ABB RobotStudio station: ProyectoFinal2021-1.rspag

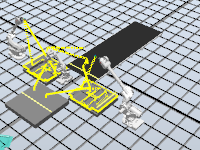
--- station ---
Station Station (saved by RobotStudio 20.4.9280.0)
Controller Controlador_Robot2, task T_ROB1: task frame (RAPID world) sits at (-153.05, 0, 0) mm in the station
Controller Controlador_Robot1, task T_ROB1: task frame (RAPID world) sits at (-2455.32, 2589.54, 0) mm in the station
Controller Controlador_PickPlace, task T_ROB1: task frame (RAPID world) sits at (-2646.21, -2443.71, 0) mm, rotated rx 0 ry 0 rz 90 deg in the station
Controller Controlador_PickPlace
  mechanical unit ROB_1: IRB6620_150_220__01, 6 joints, base frame (0, -2646.21, 459.11) mm
Controller Controlador_Robot1
  mechanical unit ROB_1: IRB7600_150_350__03, 6 joints, base frame (-2143.25, -4972.95, 0) mm
Controller Controlador_Robot2
  mechanical unit ROB_1: IRB7600_150_350__03_2, 6 joints, base frame (5003.05, -2378.13, 0) mm, rotated rx 0 ry 0 rz 180 deg
Layout (positions relative to the parent item):
  - Part Studio 3_2 [part] at (-2193.42, -2509.62, 250) mm, rotated rx 0 ry 0 rz 90 deg
  - IRB6620_150_220__01 [mechanism, from Robots\IRB6620_150_220_G_01.rslib] at (0, -2443.71, 459.11) mm, rotated rx 0 ry 0 rz 90 deg; joint values [1.5495, 0.9868, 0.0933, 0, 0.4907, -1.5921] (rad or m)
  - Vacuum Tool [mechanism] at (-1727.43, -2406.93, 788.65) mm, rotated rx 180 ry 0 rz 90 deg
      TCP tVacuum at (0, 0, 300) mm
      links: Vacuum Tool
  - Belt Conveyor [part] at (1369.01, -1300.28, 0) mm, rotated rx 0 ry 0 rz 90 deg
  - Componente inteligente_1 [smart component]
      signals: DI Attach, DI Dattach, DO Out_Sensor, DO Out_Sensor2, DO Out_Sensor22, DI AttR1, DI AttR2, DI DAttR1, DI DattR2, DO Out_Sensor5, DO Out_Sensor4, DO Out_Sensor6, DO Out_Sensor4_1, DO Out_Sensor_6_1
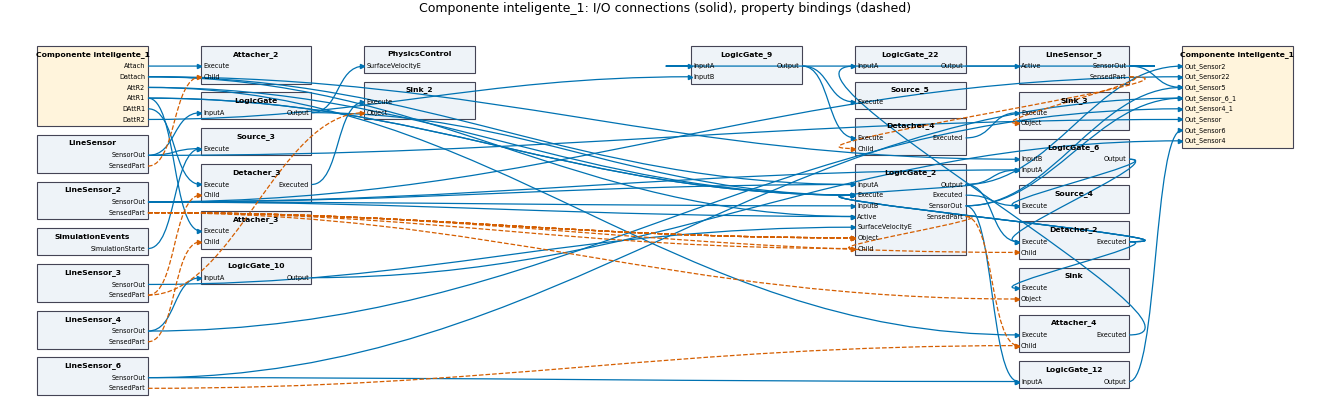
      connections:
        Componente inteligente_1.Attach -> Attacher_2.Execute
        LineSensor.SensorOut -> Source_3.Execute
        LogicGate.Output -> PhysicsControl.SurfaceVelocityEnabled
        Componente inteligente_1.Dattach -> LogicGate_2.InputA
        LogicGate_2.Output -> Detacher_2.Execute
        LogicGate.Output -> Positioner.Execute
        LineSensor_2.SensorOut -> LogicGate_3.InputB
        LogicGate_3.Output -> Positioner_2.Execute
        LogicGate_5.Output -> Componente inteligente_1.Out_Sensor2
        LineSensor_2.SensorOut -> LogicGate_5.InputA
        Detacher_2.Executed -> Positioner_3.Execute
        Detacher_2.Executed -> Positioner_4.Execute
        Componente inteligente_1.AttR2 -> Detacher_3.Execute
        Componente inteligente_1.AttR1 -> Attacher_3.Execute
        LineSensor_2.SensorOut -> Componente inteligente_1.Out_Sensor22
        Detacher_2.Executed -> Hide.Execute
        Componente inteligente_1.AttR1 -> Show.Execute
        Componente inteligente_1.Dattach -> LogicGate_6.InputB
        LogicGate_6.Output -> Detacher_2.Execute
        LineSensor_2.SensorOut -> Timer.Active
        Timer.Output -> LogicGate_6.InputA
        LineSensor_2.SensorOut -> LogicGate_6.InputA
        Hide_4.Executed -> Source_4.Execute
        Detacher_2.Executed -> Sink.Execute
        Componente inteligente_1.Dattach -> Timer_2.Active
        LogicGate_6.Output -> Source_4.Execute
        SimulationEvents.SimulationStarted -> Source_3.Execute
        Componente inteligente_1.AttR1 -> Attacher_3.Execute
        Componente inteligente_1.DAttR1 -> Detacher_3.Execute
        LineSensor_3.SensorOut -> PhysicsControl_2.SurfaceVelocityEnabled
        Detacher_3.Executed -> Sink_2.Execute
        LineSensor_5.SensorOut -> Componente inteligente_1.Out_Sensor5
        LineSensor_5.SensorOut -> Componente inteligente_1.Out_Sensor5
        LineSensor_5.SensorOut -> LogicGate_9.InputA
        Componente inteligente_1.DattR2 -> LogicGate_9.InputB
        LogicGate_9.Output -> Source_5.Execute
        LogicGate_9.Output -> Detacher_4.Execute
        Detacher_4.Executed -> Sink_3.Execute
        LineSensor_4.SensorOut -> LogicGate_10.InputA
        LineSensor_6.SensorOut -> LogicGate_12.InputA
        LineSensor_6.SensorOut -> Componente inteligente_1.Out_Sensor_6_1
        Componente inteligente_1.AttR2 -> Attacher_4.Execute
        LineSensor.SensorOut -> LogicGate.InputA
        LineSensor_6.SensorOut -> LogicGate_12.InputA
        LineSensor_6.SensorOut -> Componente inteligente_1.Out_Sensor_6_1
        LineSensor_4.SensorOut -> Componente inteligente_1.Out_Sensor4_1
        LineSensor.SensorOut -> Componente inteligente_1.Out_Sensor
        LogicGate_12.Output -> Componente inteligente_1.Out_Sensor6
        LogicGate_10.Output -> Componente inteligente_1.Out_Sensor4
        Attacher_4.Executed -> LogicGate_22.InputA
        LogicGate_22.Output -> LineSensor_5.Active
        LineSensor.SensedPart => Attacher_2.Child
        LineSensor_2.SensedPart => Detacher_2.Child
        LineSensor_2.SensedPart => Positioner.Object
        LineSensor_2.SensedPart => Positioner_2.Object
        LineSensor_2.SensedPart => Positioner_3.Object
        LineSensor_2.SensedPart => Positioner_4.Object
        LineSensor_2.SensedPart => Attacher_3.Child
        LineSensor_3.SensedPart => Detacher_3.Child
        LineSensor_2.SensedPart => Hide.Object
        LineSensor_2.SensedPart => Show.Object
        LineSensor_2.SensedPart => Sink.Object
        LineSensor_4.SensedPart => Attacher_3.Child
        LineSensor_3.SensedPart => Detacher_3.Child
        LineSensor_3.SensedPart => Sink_2.Object
        LineSensor_5.SensedPart => Detacher_4.Child
        LineSensor_5.SensedPart => Sink_3.Object
        LineSensor_6.SensedPart => Attacher_4.Child
        LineSensor_6.SensedPart => Attacher_4.Child
    - Detacher_2 [smart component, from Components\Detacher.rslib]
        properties: Child=(none); KeepPosition=true
    - Attacher_2 [smart component, from Components\Attacher.rslib]
        properties: Parent=Vacuum Tool; Flange=0; Child=(none); Mount=false; Offset=[0 0 0]; Orientation=[0 0 0]
    - LineSensor [smart component, from Components\LineSensor.rslib]
        properties: Start=[-1.2 -1 0.32]; End=[1.4 -1 0.32]; Radius=0.015; SensedPart=(none); SensedPoint=[-0.930547607421875 -1.00000006103516 0.32]
      - _sensorPart_ [part]
    - Source_3 [smart component, from Components\Source.rslib]
        properties: Source=Part Studio; Copy=(none); Parent=(none); Position=[-0.078281 5.030563 0.480363]; Orientation=[3.14159265358979 0 0]; Transient=true; PhysicsBehavior=3
    - SimulationEvents [smart component, from Components\SimulationEvents.rslib]
    - PhysicsControl [smart component, from Components\PhysicsControl.rslib]
        properties: Object=Belt Conveyor; Behavior=1; SurfaceVelocity=1
    - LogicGate [smart component, from Components\LogicGate.rslib]
        properties: Operator=NOT; Delay=0
    - LineSensor_2 [smart component, from Components\LineSensor.rslib]
        properties: Start=[-2.95 -1.5 0.533]; End=[-2.95 -3.2 0.533]; Radius=0.1; SensedPart=(none); SensedPoint=[-2.95000048828125 -1.55674926757812 0.533]
      - _sensorPart_ [part]
    - LogicGate_6 [smart component, from Components\LogicGate.rslib]
        properties: Operator=AND; Delay=1
    - Sink [smart component, from Components\Sink.rslib]
        properties: Object=(none)
    - Attacher_3 [smart component, from Components\Attacher.rslib]
        properties: Parent=Vacuum Tool; Flange=0; Child=(none); Mount=false; Offset=[0 0 0]; Orientation=[0 0 0]
    - Attacher_4 [smart component, from Components\Attacher.rslib]
        properties: Parent=Vacuum Tool; Flange=0; Child=(none); Mount=false; Offset=[0 0 0]; Orientation=[0 0 0]
    - Detacher_3 [smart component, from Components\Detacher.rslib]
        properties: Child=(none); KeepPosition=true
    - LineSensor_3 [smart component, from Components\LineSensor.rslib]
        properties: Start=[-1.2 -5 0.45]; End=[1.4 -5 0.45]; Radius=0.015; SensedPart=(none); SensedPoint=[0 0 0]
      - _sensorPart_ [part]
    - LineSensor_4 [smart component, from Components\LineSensor.rslib] at (1207.2, 0, 0) mm
        properties: Start=[-2.96159134746791 -3 0.312]; End=[-2.96159134746791 -2.881925 0.312]; Radius=0.001; SensedPart=(none); SensedPoint=[0 0 0]
      - _sensorPart_ [part]
    - Source_4 [smart component, from Components\Source.rslib]
        properties: Source=Part Studio_2; Copy=(none); Parent=(none); Position=[-1.791727 -2.471099 0.33]; Orientation=[3.14159265358979 0 1.5707963267949]; Transient=true; PhysicsBehavior=1
    - Sink_2 [smart component, from Components\Sink.rslib]
        properties: Object=(none)
    - Source_5 [smart component, from Components\Source.rslib]
        properties: Source=Part Studio_2; Copy=(none); Parent=(none); Position=[2.038141 -2.374172 0.33]; Orientation=[3.14159265358979 0 -1.5707963267949]; Transient=true; PhysicsBehavior=1
    - LineSensor_5 [smart component, from Components\LineSensor.rslib] at (6071.62, 0, 0) mm
        properties: Start=[-2.95 -1.5 0.533]; End=[-2.95 -3.2 0.533]; Radius=0.1; SensedPart=(none); SensedPoint=[0 0 0]
      - _sensorPart_ [part]
    - LogicGate_9 [smart component, from Components\LogicGate.rslib]
        properties: Operator=AND; Delay=0
    - Detacher_4 [smart component, from Components\Detacher.rslib]
        properties: Child=(none); KeepPosition=true
    - Sink_3 [smart component, from Components\Sink.rslib]
        properties: Object=(none)
    - LogicGate_10 [smart component, from Components\LogicGate.rslib]
        properties: Operator=NOT; Delay=0
    - LogicGate_12 [smart component, from Components\LogicGate.rslib]
        properties: Operator=NOT; Delay=0
    - LineSensor_6 [smart component, from Components\LineSensor.rslib] at (4964.36, 0, 0) mm
        properties: Start=[-2.96159134746791 -3 0.312]; End=[-2.96159134746791 -2.881925 0.312]; Radius=0.001; SensedPart=(none); SensedPoint=[2.0027666015625 -3 0.312]
      - _sensorPart_ [part]
    - LogicGate_22 [smart component, from Components\LogicGate.rslib]
        properties: Operator=NOT; Delay=0
  - Part Studio [part] at (384.19, -4809.35, 381.64) mm, rotated rx 180 ry 0 rz 0 deg
  - IRB7600_150_350__03 [mechanism, from Robots\IRB7600_150_350_G_03.rslib] at (-4598.56, -2383.41, 0) mm; joint values [0, -0.9152, 0, 0, 0.5236, 0] (rad or m)
  - LogicGate_7 [smart component, from Components\LogicGate.rslib]
      properties: Operator=AND; Delay=0
  - Pieza_1 [part] at (-1268.57, -2175.31, 0) mm
  - HerramientaDeCorte [mechanism, from Libraries\HerramientaDeCorte.rslib] at (-3713.92, -2383.41, 3226.26) mm, rotated rx 0 ry 67.56 rz 0 deg
  - Part Studio_2 [part] at (2038.14, -2374.17, 330) mm, rotated rx 180 ry 0 rz -90 deg
  - Part Studio 3_3 [part] at (2439.83, -2335.65, 250) mm, rotated rx 0 ry 0 rz -90 deg
  - IRB7600_150_350__03_2 [mechanism, from Robots\IRB7600_150_350_G_03.rslib] at (4850, -2378.13, 0) mm, rotated rx 0 ry 0 rz 180 deg; joint values [0, 0, -0.648, 0, 0.5236, 0] (rad or m)
  - HerramientaDeCorte_2 [mechanism, from Libraries\HerramientaDeCorte_1.rslib] at (2687.31, -2378.13, 3231.92) mm, rotated rx 0 ry 82.87 rz 180 deg
  - LogicGate_8 [smart component, from Components\LogicGate.rslib]
      properties: Operator=AND; Delay=0
  - LogicGate_11 [smart component, from Components\LogicGate.rslib]
      properties: Operator=AND; Delay=0
  - LogicGate_13 [smart component, from Components\LogicGate.rslib]
      properties: Operator=AND; Delay=0
  - LogicGate_14 [smart component, from Components\LogicGate.rslib]
      properties: Operator=AND; Delay=0
  - LogicGate_15 [smart component, from Components\LogicGate.rslib]
      properties: Operator=AND; Delay=0
  - LogicGate_16 [smart component, from Components\LogicGate.rslib]
      properties: Operator=AND; Delay=0
  - LogicGate_17 [smart component, from Components\LogicGate.rslib]
      properties: Operator=AND; Delay=0
  - LogicGate_18 [smart component, from Components\LogicGate.rslib]
      properties: Operator=AND; Delay=0
  - LogicGate_19 [smart component, from Components\LogicGate.rslib]
      properties: Operator=NOT; Delay=0
  - LogicGate_20 [smart component, from Components\LogicGate.rslib]
      properties: Operator=AND; Delay=0
  - LogicGate_21 [smart component, from Components\LogicGate.rslib]
      properties: Operator=NOT; Delay=0
  - Part Studio_291 [part] at (700.63, -8575.01, 80.62) mm, rotated rx -178.41 ry 0 rz 123.64 deg
Attachment: Vacuum Tool is attached to IRB6620_150_220__01 / Link6
Attachment: HerramientaDeCorte is attached to IRB7600_150_350__03 / Link6
Attachment: HerramientaDeCorte_2 is attached to IRB7600_150_350__03_2 / Link6
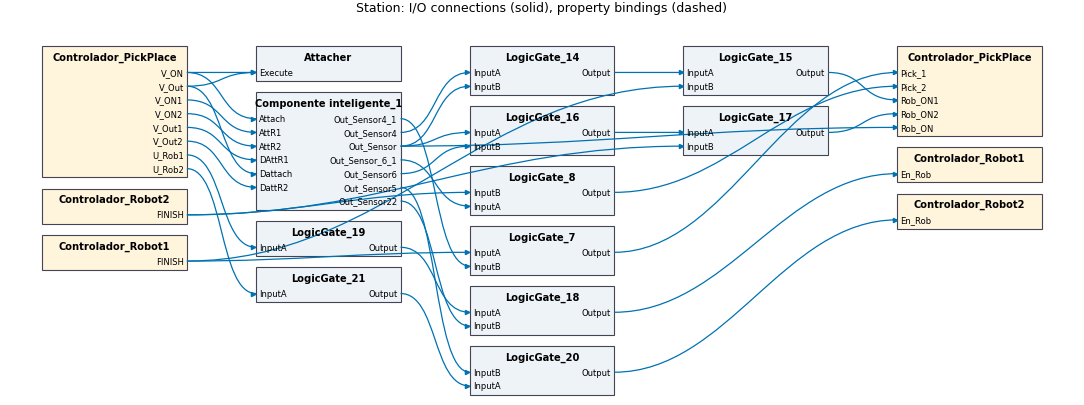
Station logic (signal -> signal, property => property):
  Controlador_PickPlace.V_ON -> Attacher.Execute
  Controlador_PickPlace.V_Out -> Detacher.Execute
  Controlador_PickPlace.V_ON -> Componente inteligente_1.Attach
  Controlador_PickPlace.V_ON1 -> Componente inteligente_1.AttR1
  Controlador_PickPlace.V_ON2 -> Componente inteligente_1.AttR2
  Controlador_PickPlace.V_Out1 -> Componente inteligente_1.DAttR1
  Controlador_PickPlace.V_Out -> Componente inteligente_1.Dattach
  Controlador_Robot2.FINISH -> LogicGate_8.InputB
  Controlador_PickPlace.V_Out2 -> Componente inteligente_1.DattR2
  Controlador_Robot1.FINISH -> LogicGate_7.InputA
  Componente inteligente_1.Out_Sensor4_1 -> LogicGate_7.InputB
  Componente inteligente_1.Out_Sensor4 -> LogicGate_14.InputA
  Componente inteligente_1.Out_Sensor -> LogicGate_14.InputB
  LogicGate_14.Output -> LogicGate_15.InputA
  Controlador_Robot1.FINISH -> LogicGate_15.InputB
  LogicGate_7.Output -> Controlador_PickPlace.Pick_1
  Componente inteligente_1.Out_Sensor_6_1 -> LogicGate_8.InputA
  LogicGate_8.Output -> Controlador_PickPlace.Pick_2
  Componente inteligente_1.Out_Sensor -> LogicGate_16.InputA
  Componente inteligente_1.Out_Sensor6 -> LogicGate_16.InputB
  LogicGate_16.Output -> LogicGate_17.InputA
  Controlador_Robot2.FINISH -> LogicGate_17.InputB
  LogicGate_15.Output -> Controlador_PickPlace.Rob_ON1
  LogicGate_17.Output -> Controlador_PickPlace.Rob_ON2
  Componente inteligente_1.Out_Sensor -> Controlador_PickPlace.Rob_ON
  Controlador_PickPlace.U_Rob1 -> LogicGate_19.InputA
  LogicGate_19.Output -> LogicGate_18.InputA
  LogicGate_18.Output -> Controlador_Robot1.En_Rob
  Controlador_PickPlace.U_Rob2 -> LogicGate_21.InputA
  Componente inteligente_1.Out_Sensor5 -> LogicGate_20.InputB
  LogicGate_21.Output -> LogicGate_20.InputA
  LogicGate_20.Output -> Controlador_Robot2.En_Rob
  Componente inteligente_1.Out_Sensor22 -> LogicGate_18.InputB
Targets, tools, work objects and paths stored in the station and not in the controller backup, written as RAPID:
! task T_ROB1
MODULE Module1
  CONST robtarget Target_274:=[[250.928875654,-5796.464620021,317.65],[0,-0.707106781,0.707106781,0],[-1,0,-2,0],[9E+09,9E+09,9E+09,9E+09,9E+09,9E+09]];
  CONST robtarget Target_404:=[[700.928875654,-5166.464620021,352.65],[0,-0.707106781,0.707106781,0],[-1,0,-2,0],[9E+09,9E+09,9E+09,9E+09,9E+09,9E+09]];
  CONST robtarget Target_444:=[[700.928875654,-4846.464620021,352.65],[0,-0.707106781,0.707106781,0],[0,0,-1,0],[9E+09,9E+09,9E+09,9E+09,9E+09,9E+09]];
ENDMODULE


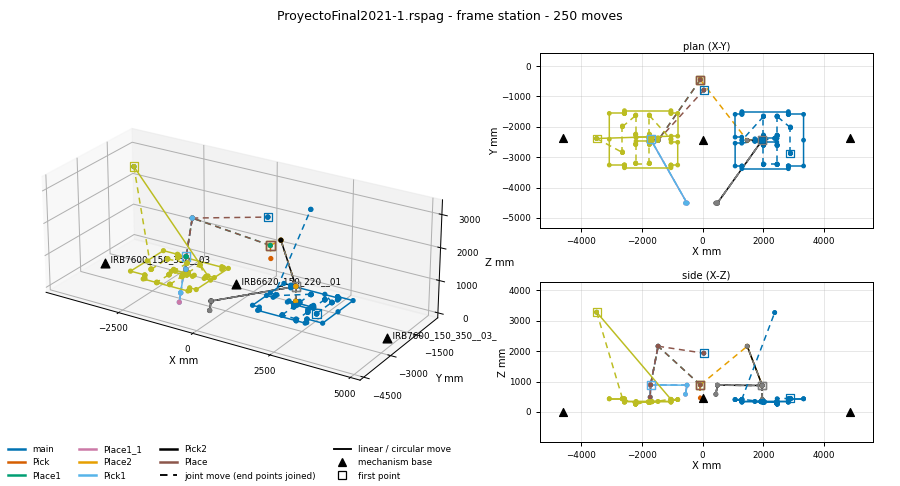
[picture p0: tool path of ProyectoFinal2021-1.rspag in frame station, 250 of 250 moves have a stored position in this frame; points joined in program order, loops and branches not executed]
--- Backups/Controlador_PickPlace/RAPID/TASK1/PROGMOD/CalibData.mod ---
MODULE CalibData
    PERS tooldata tVacuum:=[TRUE,[[0,0,300],[1,0,0,0]],[11,[0,0,200],[1,0,0,0],0,0,0]];
ENDMODULE

--- Backups/Controlador_PickPlace/RAPID/TASK1/PROGMOD/Module1.mod ---
MODULE Module1
        CONST robtarget Target_10:=[[0,-1179.406420384,2164.113508615],[0.353553391,-0.612372436,0.612372436,0.353553391],[0,-1,0,0],[9E+09,9E+09,9E+09,9E+09,9E+09,9E+09]];
    CONST robtarget Target_20_2:=[[1993.099436165,-2567.929041541,890],[0,-0.707106781,0.707106781,0],[-1,0,-1,0],[9E+09,9E+09,9E+09,9E+09,9E+09,9E+09]];
    CONST robtarget Target_20:=[[2025.267436165,-2567.931041541,460.348],[0,-0.707106781,0.707106781,0],[-2,0,-2,0],[9E+09,9E+09,9E+09,9E+09,9E+09,9E+09]];
    CONST robtarget Target_30_2:=[[36.785436165,-931.826041541,890],[0,1,0,0],[-1,0,-2,0],[9E+09,9E+09,9E+09,9E+09,9E+09,9E+09]];
    CONST robtarget Target_30:=[[36.785436165,-918.776041541,488.65],[0,1,0,0],[-1,0,-2,0],[9E+09,9E+09,9E+09,9E+09,9E+09,9E+09]];
    CONST robtarget Target_30_3:=[[2015.725,-2164.754477706,320.279],[0,-0.707106781,0.707106781,0],[0,0,-1,0],[9E+09,9E+09,9E+09,9E+09,9E+09,9E+09]];
    CONST robtarget Target_40:=[[-2065.640563835,-2080.403041541,581.641],[0,-0.707106781,0.707106781,0],[0,0,0,0],[9E+09,9E+09,9E+09,9E+09,9E+09,9E+09]];
    CONST robtarget Target_50:=[[5.364436165,-4607.016041541,411.65],[0,0,1,0],[-1,0,-1,0],[9E+09,9E+09,9E+09,9E+09,9E+09,9E+09]];
    CONST robtarget Target_60:=[[0,-4113.021984806,2164.113532469],[0.353553384,0.612372439,0.612372439,-0.353553384],[-2,0,-1,0],[9E+09,9E+09,9E+09,9E+09,9E+09,9E+09]];
    CONST robtarget Target_70:=[[1653.263,-2683.789477706,1934.535],[0,-0.707106781,0.707106781,0],[-1,0,-2,0],[9E+09,9E+09,9E+09,9E+09,9E+09,9E+09]];
    CONST robtarget Target_80:=[[-2065.640563835,-3080.403041541,581.641],[0,1,0,0],[-2,0,-1,0],[9E+09,9E+09,9E+09,9E+09,9E+09,9E+09]];
    CONST robtarget Target_90:=[[1653.26,-2638.786477706,434.509],[0,-0.707106781,0.707106781,0],[0,0,-1,0],[9E+09,9E+09,9E+09,9E+09,9E+09,9E+09]];
    CONST robtarget Target_100:=[[1553.362,-2638.786477706,441.414],[0,-0.707106781,0.707106781,0],[0,0,-1,0],[9E+09,9E+09,9E+09,9E+09,9E+09,9E+09]];
    CONST robtarget Target_110:=[[1453.462,-2638.788477706,448.319],[0,-0.707106781,0.707106781,0],[0,0,-1,0],[9E+09,9E+09,9E+09,9E+09,9E+09,9E+09]];
    CONST robtarget Target_120:=[[1453.471,-2728.784477706,448.368],[0,-0.707106781,0.707106781,0],[-1,0,-2,0],[9E+09,9E+09,9E+09,9E+09,9E+09,9E+09]];
    CONST robtarget Target_40_2:=[[-2065.640563835,-2130.403041541,881.641],[0,-0.707106781,0.707106781,0],[0,0,0,0],[9E+09,9E+09,9E+09,9E+09,9E+09,9E+09]];
    CONST robtarget Target_50_2:=[[5.364436165,-4607.016041541,871.65],[0,0,1,0],[-1,0,-1,0],[9E+09,9E+09,9E+09,9E+09,9E+09,9E+09]];
    CONST robtarget Target_80_2:=[[-2065.640563835,-3130.403041541,881.641],[0,1,0,0],[-2,0,-1,0],[9E+09,9E+09,9E+09,9E+09,9E+09,9E+09]];
!***********************************************************
    !
    ! Módulo:  Module1
    !
    ! Descripción:
    !   <Introduzca la descripción aquí>
    !
    ! Autor: Alex
    !
    ! Versión: 1.0
    !
    !***********************************************************


    !***********************************************************
    !
    ! Procedimiento Main
    !
    !   Este es el punto de entrada de su programa
    !
    !***********************************************************
    PROC main()
        Init:
        SetDO V_Out,0;
        SetDO V_ON,0;
        SetDO U_Rob1,0;
        SetDO U_Rob2,0;
        MoveJ Target_70,v1000,z100,tVacuum\WObj:=wobj0;
        WaitDI Rob_ON,1;
 !       WaitUntil Rob_ON1=1 OR Rob_ON2=1 OR Pick_1=1 OR Pick_2=1 OR Rob_ON1=0 OR Rob_ON2=0 OR Pick_1=0 OR Pick_2=0;
        IF Rob_ON1=1 THEN ! Detecta si robot está quieto, hay tapete esperando y no hay tapete en estación 1, pone tapete en estación 1
           pick;
           place1;
        ELSEIF Rob_ON2=1 THEN ! Detecta si robot está quieto, hay tapete esperando y no hay tapete en estación 2, pone tapete en estación 2
           pick;
           place2;
        ELSEIF Pick_1=1 THEN !Detecta si robot 1 está quieto y hay tapete en estación 1, lleva el tapete de estación 1 a mesa
           pick1;
        ELSEIF Pick_2=1 THEN !Detecta si robot 2 está quieto y hay tapete en estación 2, lleva el tapete de estación 2 a mesa
           pick2;
        ELSE MoveJ Target_70,v1000,fine,tVacuum\WObj:=wobj0;
        ENDIF
        GOTO Init;
        !Añada aquí su código
    ENDPROC
    PROC Pick()
        MoveJ Target_20_2,v1000,fine,tVacuum\WObj:=wobj0;
        MoveJ Target_20,v1000,fine,tVacuum\WObj:=wobj0;
        WaitTime 1;
        SetDO V_ON,1;
        WaitTime 2;
        SetDO V_ON,0;
    ENDPROC
    PROC Place1()
        MoveJ Target_20_2,v1000,fine,tVacuum\WObj:=wobj0;
        MoveJ Target_10,v1000,fine,tVacuum\WObj:=wobj0;
        MoveJ Target_30_2,v1000,fine,tVacuum\WObj:=wobj0;
        MoveJ Target_30,v1000,fine,tVacuum\WObj:=wobj0;
        WaitTime 1;
        SetDO V_Out,1;
        WaitTime 1;
        SetDO V_Out,0;
        MoveJ Target_30_2,v1000,fine,tVacuum\WObj:=wobj0;
        MoveJ Target_10,v1000,fine,tVacuum\WObj:=wobj0;
    ENDPROC
    PROC Place1_1()
        MoveJ Target_30_2,v1000,fine,tVacuum\WObj:=wobj0;
        WaitTime 1;
        MoveJ Target_30,v1000,fine,tVacuum\WObj:=wobj0;
        SetDO V_ON1,1;
        WaitTime 1;
        SetDO V_ON1,0;
        MoveJ Target_30_2,v1000,fine,tVacuum\WObj:=wobj0;
        MoveJ Target_40_2,v1000,fine,tVacuum\WObj:=wobj0;
        MoveJ Target_40,v1000,fine,tVacuum\WObj:=wobj0;
        SetDO V_Out1,1;
        WaitTime 1;
        SetDO V_Out1,0;
        MoveJ Target_40_2,v1000,fine,tVacuum\WObj:=wobj0;
        MoveJ Target_30_2,v1000,fine,tVacuum\WObj:=wobj0;
        MoveJ Target_10,v1000,fine,tVacuum\WObj:=wobj0;
    ENDPROC
    PROC Place2()
        MoveJ Target_20_2,v1000,fine,tVacuum\WObj:=wobj0;
        MoveJ Target_60,v1000,fine,tVacuum\WObj:=wobj0;
        MoveJ Target_50_2,v1000,fine,tVacuum\WObj:=wobj0;
        WaitTime 1;
        MoveJ Target_50,v1000,fine,tVacuum\WObj:=wobj0;
        WaitTime 1;
        SetDO V_Out2,1;
        WaitTime 1;
        SetDO V_Out2,0;
        MoveJ Target_50_2,v1000,fine,tVacuum\WObj:=wobj0;
        MoveJ Target_60,v1000,fine,tVacuum\WObj:=wobj0;
    ENDPROC
    PROC Pick1()
        MoveL Target_30_2,v1000,fine,tVacuum\WObj:=wobj0;
        MoveL Target_30,v1000,fine,tVacuum\WObj:=wobj0;
        SetDO V_ON1,1;
        WaitTime 2;
        SetDO V_ON1,0;
        SetDO U_Rob1,1;
        MoveL Target_30_2,v1000,fine,tVacuum\WObj:=wobj0;
        MoveL Target_40_2,v1000,fine,tVacuum\WObj:=wobj0;
        MoveL Target_40,v1000,fine,tVacuum\WObj:=wobj0;
        SetDO V_Out1,1;
        WaitTime 2;
        SetDO V_Out1,0;
        WaitTime 2;
        SetDO U_Rob1,0;
        MoveJ Target_40_2,v1000,fine,tVacuum\WObj:=wobj0;
        MoveJ Target_30_2,v1000,fine,tVacuum\WObj:=wobj0;
        MoveJ Target_10,v1000,fine,tVacuum\WObj:=wobj0;
    ENDPROC
    PROC Pick2()
        MoveJ Target_50_2,v1000,fine,tVacuum\WObj:=wobj0;
        MoveJ Target_50,v1000,fine,tVacuum\WObj:=wobj0;
        SetDO V_ON2,1;
        WaitTime 2;
        SetDO V_ON2,0;
        WaitTime 2;
        SetDO U_Rob2,1;
        MoveJ Target_50_2,v1000,fine,tVacuum\WObj:=wobj0;
        MoveJ Target_80_2,v1000,fine,tVacuum\WObj:=wobj0;
        MoveJ Target_80,v1000,fine,tVacuum\WObj:=wobj0;
        SetDO V_Out1,1;
        WaitTime 2;
        SetDO V_Out1,0;
        WaitTime 2;
        SetDO U_Rob2,0;
        MoveL Target_80_2,v1000,fine,tVacuum\WObj:=wobj0;
        MoveL Target_50_2,v1000,fine,tVacuum\WObj:=wobj0;
        MoveL Target_60,v1000,fine,tVacuum\WObj:=wobj0;
    ENDPROC
    PROC Place()
        MoveJ Target_20_2,v1000,fine,tVacuum\WObj:=wobj0;
        MoveJ Target_10,v1000,fine,tVacuum\WObj:=wobj0;
        MoveJ Target_30_2,v1000,fine,tVacuum\WObj:=wobj0;
        MoveJ Target_30,v1000,fine,tVacuum\WObj:=wobj0;
        WaitTime 1;
        SetDO V_Out,1;
        WaitTime 1;
        SetDO V_Out,0;
        MoveJ Target_30_2,v1000,fine,tVacuum\WObj:=wobj0;
        MoveJ Target_10,v1000,fine,tVacuum\WObj:=wobj0;
        MoveJ Target_70,v1000,fine,tVacuum\WObj:=wobj0;
    ENDPROC
    PROC Place2_1()
        MoveJ Target_50_2,v1000,fine,tVacuum\WObj:=wobj0;
        MoveJ Target_50,v1000,fine,tVacuum\WObj:=wobj0;
        SetDO V_ON2,1;
        WaitTime 2;
        SetDO V_ON2,0;
        MoveJ Target_50_2,v1000,fine,tVacuum\WObj:=wobj0;
        MoveJ Target_80_2,v1000,fine,tVacuum\WObj:=wobj0;
        MoveJ Target_80,v1000,fine,tVacuum\WObj:=wobj0;
        SetDO V_out1,1;
        WaitTime 2;
        SetDO V_Out1,0;
        MoveJ Target_80_2,v1000,fine,tVacuum\WObj:=wobj0;
        MoveJ Target_50_2,v1000,fine,tVacuum\WObj:=wobj0;
        MoveJ Target_60,v1000,fine,tVacuum\WObj:=wobj0;
    ENDPROC

ENDMODULE

--- Backups/Controlador_Robot1/RAPID/TASK1/PROGMOD/CalibData.mod ---
MODULE CalibData
    PERS tooldata MyTool:=[TRUE,[[31.7926,0,229.639],[0.945519,0,0.325568,0]],[1,[0,0,1],[1,0,0,0],0,0,0]];
    PERS tooldata HerramientaDeCorte:=[TRUE,[[0,0,319.427],[1,0,0,0]],[1,[0,0,1],[1,0,0,0],0,0,0]];
ENDMODULE

--- Backups/Controlador_Robot1/RAPID/TASK1/PROGMOD/Module1.mod ---
MODULE Module1
        CONST robtarget Target_10:=[[783.928875653,-4994.669620021,486.089],[0,-0.707106781,0.707106781,0],[0,0,0,0],[9E+09,9E+09,9E+09,9E+09,9E+09,9E+09]];
    CONST robtarget Target_20:=[[740.928875653,-4996.464620021,391.65],[0,-0.707106781,0.707106781,0],[0,0,-1,0],[9E+09,9E+09,9E+09,9E+09,9E+09,9E+09]];
    CONST robtarget Target_10_2:=[[783.928875653,-4994.669620021,936.089],[0,-0.707106781,0.707106781,0],[0,0,-1,0],[9E+09,9E+09,9E+09,9E+09,9E+09,9E+09]];
    CONST robtarget Target_30:=[[-1034.222247941,-4972.95221081,3284.527172221],[0.604871201,0,0.79632332,0],[-1,0,-1,0],[9E+09,9E+09,9E+09,9E+09,9E+09,9E+09]];
    CONST robtarget Target_20_3:=[[740.928875653,-4996.464620021,451.65],[0,-0.707106781,0.707106781,0],[0,0,-1,0],[9E+09,9E+09,9E+09,9E+09,9E+09,9E+09]];
        TASK PERS tooldata tool1:=[TRUE,[[0,0,0],[1,0,0,0]],[-1,[0,0,0],[1,0,0,0],0,0,0]];
    CONST robtarget Target_35:=[[-186.231124346,-5433.964620021,446.65],[0,-0.707106781,0.707106781,0],[-1,0,-2,0],[9E+09,9E+09,9E+09,9E+09,9E+09,9E+09]];
    CONST robtarget Target_40:=[[-186.231124346,-5433.964620021,432.65],[0,-0.707106781,0.707106781,0],[-1,0,-2,0],[9E+09,9E+09,9E+09,9E+09,9E+09,9E+09]];
    CONST robtarget Target_50:=[[-173.731124346,-5421.464620021,432.65],[0,-0.707106781,0.707106781,0],[-1,0,-2,0],[9E+09,9E+09,9E+09,9E+09,9E+09,9E+09]];
    CONST robtarget Target_60:=[[-186.231124346,-5408.964620021,432.65],[0,-0.707106781,0.707106781,0],[-1,0,-2,0],[9E+09,9E+09,9E+09,9E+09,9E+09,9E+09]];
    CONST robtarget Target_70:=[[-198.731124346,-5421.464620021,432.65],[0,-0.707106781,0.707106781,0],[-1,0,-2,0],[9E+09,9E+09,9E+09,9E+09,9E+09,9E+09]];
    CONST robtarget Target_90:=[[-173.731124346,-4571.464620021,432.65],[0,-0.707106781,0.707106781,0],[0,0,0,0],[9E+09,9E+09,9E+09,9E+09,9E+09,9E+09]];
    CONST robtarget Target_110:=[[-198.731124346,-4571.464620021,432.65],[0,-0.707106781,0.707106781,0],[0,0,0,0],[9E+09,9E+09,9E+09,9E+09,9E+09,9E+09]];
    CONST robtarget Target_114:=[[250.928875654,-4216.464620021,437.65],[0,-0.707106781,0.707106781,0],[0,0,-1,0],[9E+09,9E+09,9E+09,9E+09,9E+09,9E+09]];
    CONST robtarget Target_115:=[[250.928875654,-4216.464620021,277.65],[0,-0.707106781,0.707106781,0],[0,0,0,0],[9E+09,9E+09,9E+09,9E+09,9E+09,9E+09]];
    CONST robtarget Target_120:=[[250.928875654,-4216.464620021,262.65],[0,-0.707106781,0.707106781,0],[0,0,0,0],[9E+09,9E+09,9E+09,9E+09,9E+09,9E+09]];
    CONST robtarget Target_130:=[[260.928875654,-4206.464620021,262.65],[0,-0.707106781,0.707106781,0],[0,0,0,0],[9E+09,9E+09,9E+09,9E+09,9E+09,9E+09]];
    CONST robtarget Target_140:=[[250.928875654,-4196.464620021,262.65],[0,-0.707106781,0.707106781,0],[0,0,0,0],[9E+09,9E+09,9E+09,9E+09,9E+09,9E+09]];
    CONST robtarget Target_150:=[[240.928875654,-4206.464620021,262.65],[0,-0.707106781,0.707106781,0],[0,0,0,0],[9E+09,9E+09,9E+09,9E+09,9E+09,9E+09]];
    CONST robtarget Target_155:=[[250.928875654,-4846.464620021,277.65],[0,-0.707106781,0.707106781,0],[0,0,0,0],[9E+09,9E+09,9E+09,9E+09,9E+09,9E+09]];
    CONST robtarget Target_160:=[[250.928875654,-4846.464620021,262.65],[0,-0.707106781,0.707106781,0],[0,0,0,0],[9E+09,9E+09,9E+09,9E+09,9E+09,9E+09]];
    CONST robtarget Target_170:=[[260.928875654,-4836.464620021,262.65],[0,-0.707106781,0.707106781,0],[0,0,0,0],[9E+09,9E+09,9E+09,9E+09,9E+09,9E+09]];
    CONST robtarget Target_180:=[[250.928875654,-4826.464620021,262.65],[0,-0.707106781,0.707106781,0],[0,0,0,0],[9E+09,9E+09,9E+09,9E+09,9E+09,9E+09]];
    CONST robtarget Target_190:=[[240.928875654,-4836.464620021,262.65],[0,-0.707106781,0.707106781,0],[0,0,0,0],[9E+09,9E+09,9E+09,9E+09,9E+09,9E+09]];
    CONST robtarget Target_195:=[[261.901875654,-4932.290620021,347.65],[0,-0.707106781,0.707106781,0],[0,0,0,0],[9E+09,9E+09,9E+09,9E+09,9E+09,9E+09]];
    CONST robtarget Target_200:=[[261.901875654,-4932.290620021,332.65],[0,-0.707106781,0.707106781,0],[0,0,0,0],[9E+09,9E+09,9E+09,9E+09,9E+09,9E+09]];
    CONST robtarget Target_210:=[[261.901875654,-5060.638620021,332.65],[0,-0.707106781,0.707106781,0],[-1,0,-2,0],[9E+09,9E+09,9E+09,9E+09,9E+09,9E+09]];
    CONST robtarget Target_220:=[[663.589875654,-5060.638620021,332.65],[0,-0.707106781,0.707106781,0],[-1,0,-2,0],[9E+09,9E+09,9E+09,9E+09,9E+09,9E+09]];
    CONST robtarget Target_230:=[[663.589875654,-4932.290620021,332.65],[0,-0.707106781,0.707106781,0],[0,0,0,0],[9E+09,9E+09,9E+09,9E+09,9E+09,9E+09]];
    CONST robtarget Target_234:=[[250.928875654,-5166.464620021,362.65],[0,-0.707106781,0.707106781,0],[-1,0,-2,0],[9E+09,9E+09,9E+09,9E+09,9E+09,9E+09]];
    CONST robtarget Target_235:=[[250.928875654,-5166.464620021,277.65],[0,-0.707106781,0.707106781,0],[-1,0,-2,0],[9E+09,9E+09,9E+09,9E+09,9E+09,9E+09]];
    CONST robtarget Target_240:=[[250.928875654,-5166.464620021,262.65],[0,-0.707106781,0.707106781,0],[-1,0,-2,0],[9E+09,9E+09,9E+09,9E+09,9E+09,9E+09]];
    CONST robtarget Target_250:=[[260.928875654,-5156.464620021,262.65],[0,-0.707106781,0.707106781,0],[-1,0,-2,0],[9E+09,9E+09,9E+09,9E+09,9E+09,9E+09]];
    CONST robtarget Target_260:=[[250.928875654,-5146.464620021,262.65],[0,-0.707106781,0.707106781,0],[-1,0,-2,0],[9E+09,9E+09,9E+09,9E+09,9E+09,9E+09]];
    CONST robtarget Target_270:=[[240.928875654,-5156.464620021,262.65],[0,-0.707106781,0.707106781,0],[-1,0,-2,0],[9E+09,9E+09,9E+09,9E+09,9E+09,9E+09]];
    CONST robtarget Target_275:=[[250.928875654,-5796.464620021,277.65],[0,-0.707106781,0.707106781,0],[-1,0,-2,0],[9E+09,9E+09,9E+09,9E+09,9E+09,9E+09]];
    CONST robtarget Target_280:=[[250.928875654,-5796.464620021,262.65],[0,-0.707106781,0.707106781,0],[-1,0,-2,0],[9E+09,9E+09,9E+09,9E+09,9E+09,9E+09]];
    CONST robtarget Target_290:=[[260.928875654,-5786.464620021,262.65],[0,-0.707106781,0.707106781,0],[-1,0,-2,0],[9E+09,9E+09,9E+09,9E+09,9E+09,9E+09]];
    CONST robtarget Target_300:=[[250.928875654,-5776.464620021,262.65],[0,-0.707106781,0.707106781,0],[-1,0,-2,0],[9E+09,9E+09,9E+09,9E+09,9E+09,9E+09]];
    CONST robtarget Target_310:=[[240.928875654,-5786.464620021,262.65],[0,-0.707106781,0.707106781,0],[-1,0,-2,0],[9E+09,9E+09,9E+09,9E+09,9E+09,9E+09]];
    CONST robtarget Target_325:=[[700.928875654,-5796.464620021,327.65],[0,-0.707106781,0.707106781,0],[-1,0,-2,0],[9E+09,9E+09,9E+09,9E+09,9E+09,9E+09]];
    CONST robtarget Target_330:=[[700.928875654,-5796.464620021,312.65],[0,-0.707106781,0.707106781,0],[-1,0,-2,0],[9E+09,9E+09,9E+09,9E+09,9E+09,9E+09]];
    CONST robtarget Target_340:=[[710.928875654,-5786.464620021,312.65],[0,-0.707106781,0.707106781,0],[-1,0,-2,0],[9E+09,9E+09,9E+09,9E+09,9E+09,9E+09]];
    CONST robtarget Target_350:=[[700.928875654,-5776.464620021,312.65],[0,-0.707106781,0.707106781,0],[-1,0,-2,0],[9E+09,9E+09,9E+09,9E+09,9E+09,9E+09]];
    CONST robtarget Target_360:=[[690.928875654,-5786.464620021,312.65],[0,-0.707106781,0.707106781,0],[-1,0,-2,0],[9E+09,9E+09,9E+09,9E+09,9E+09,9E+09]];
    CONST robtarget Target_365:=[[700.928875654,-5166.464620021,327.65],[0,-0.707106781,0.707106781,0],[-1,0,-2,0],[9E+09,9E+09,9E+09,9E+09,9E+09,9E+09]];
    CONST robtarget Target_370:=[[700.928875654,-5166.464620021,312.65],[0,-0.707106781,0.707106781,0],[-1,0,-2,0],[9E+09,9E+09,9E+09,9E+09,9E+09,9E+09]];
    CONST robtarget Target_380:=[[710.928875654,-5156.464620021,312.65],[0,-0.707106781,0.707106781,0],[-1,0,-2,0],[9E+09,9E+09,9E+09,9E+09,9E+09,9E+09]];
    CONST robtarget Target_390:=[[700.928875654,-5146.464620021,312.65],[0,-0.707106781,0.707106781,0],[-1,0,-2,0],[9E+09,9E+09,9E+09,9E+09,9E+09,9E+09]];
    CONST robtarget Target_400:=[[690.928875654,-5156.464620021,312.65],[0,-0.707106781,0.707106781,0],[-1,0,-2,0],[9E+09,9E+09,9E+09,9E+09,9E+09,9E+09]];
    CONST robtarget Target_405:=[[783.642875654,-5041.464620021,349.902],[0,-0.707106781,0.707106781,0],[-1,0,-2,0],[9E+09,9E+09,9E+09,9E+09,9E+09,9E+09]];
    CONST robtarget Target_410:=[[783.642875654,-5041.464620021,334.902],[0,-0.707106781,0.707106781,0],[-1,0,-2,0],[9E+09,9E+09,9E+09,9E+09,9E+09,9E+09]];
    CONST robtarget Target_420:=[[983.642875654,-5041.464620021,345.449],[0,-0.707106781,0.707106781,0],[-1,0,-2,0],[9E+09,9E+09,9E+09,9E+09,9E+09,9E+09]];
    CONST robtarget Target_430:=[[983.642875654,-4951.464620021,345.449],[0,-0.707106781,0.707106781,0],[0,0,0,0],[9E+09,9E+09,9E+09,9E+09,9E+09,9E+09]];
    CONST robtarget Target_440:=[[783.642875654,-4951.464620021,334.902],[0,-0.707106781,0.707106781,0],[0,0,0,0],[9E+09,9E+09,9E+09,9E+09,9E+09,9E+09]];
    CONST robtarget Target_445:=[[700.928875654,-4846.464620021,327.65],[0,-0.707106781,0.707106781,0],[0,0,0,0],[9E+09,9E+09,9E+09,9E+09,9E+09,9E+09]];
    CONST robtarget Target_450:=[[700.928875654,-4846.464620021,312.65],[0,-0.707106781,0.707106781,0],[0,0,0,0],[9E+09,9E+09,9E+09,9E+09,9E+09,9E+09]];
    CONST robtarget Target_460:=[[710.928875654,-4836.464620021,312.65],[0,-0.707106781,0.707106781,0],[0,0,0,0],[9E+09,9E+09,9E+09,9E+09,9E+09,9E+09]];
    CONST robtarget Target_470:=[[700.928875654,-4826.464620021,312.65],[0,-0.707106781,0.707106781,0],[0,0,0,0],[9E+09,9E+09,9E+09,9E+09,9E+09,9E+09]];
    CONST robtarget Target_480:=[[690.928875654,-4836.464620021,312.65],[0,-0.707106781,0.707106781,0],[0,0,0,0],[9E+09,9E+09,9E+09,9E+09,9E+09,9E+09]];
    CONST robtarget Target_485:=[[700.928875654,-4216.464620021,327.65],[0,-0.707106781,0.707106781,0],[0,0,0,0],[9E+09,9E+09,9E+09,9E+09,9E+09,9E+09]];
    CONST robtarget Target_490:=[[700.928875654,-4216.464620021,312.65],[0,-0.707106781,0.707106781,0],[0,0,0,0],[9E+09,9E+09,9E+09,9E+09,9E+09,9E+09]];
    CONST robtarget Target_500:=[[710.928875654,-4206.464620021,312.65],[0,-0.707106781,0.707106781,0],[0,0,0,0],[9E+09,9E+09,9E+09,9E+09,9E+09,9E+09]];
    CONST robtarget Target_510:=[[700.928875654,-4196.464620021,312.65],[0,-0.707106781,0.707106781,0],[0,0,0,0],[9E+09,9E+09,9E+09,9E+09,9E+09,9E+09]];
    CONST robtarget Target_520:=[[690.928875654,-4206.464620021,312.65],[0,-0.707106781,0.707106781,0],[0,0,0,0],[9E+09,9E+09,9E+09,9E+09,9E+09,9E+09]];
    CONST robtarget Target_530:=[[-963.36800286,-4972.95221081,3348.184668964],[0.831174335,0,0.556011892,0],[-1,0,-1,0],[9E+09,9E+09,9E+09,9E+09,9E+09,9E+09]];
    CONST robtarget Target_194:=[[240.928875654,-4836.464620021,347.65],[0,-0.707106781,0.707106781,0],[0,0,-1,0],[9E+09,9E+09,9E+09,9E+09,9E+09,9E+09]];
    CONST robtarget Target_75:=[[-186.231124346,-4583.964620021,446.65],[0,-0.707106781,0.707106781,0],[0,0,-1,0],[9E+09,9E+09,9E+09,9E+09,9E+09,9E+09]];
    CONST robtarget Target_100:=[[-186.231124346,-4558.964620021,432.65],[0,-0.707106781,0.707106781,0],[0,0,0,0],[9E+09,9E+09,9E+09,9E+09,9E+09,9E+09]];
    CONST robtarget Target_80:=[[-186.231124346,-4583.964620021,432.65],[0,-0.707106781,0.707106781,0],[0,0,-1,0],[9E+09,9E+09,9E+09,9E+09,9E+09,9E+09]];
    CONST robtarget Target_535:=[[1402.542526463,-4996.464620021,420.778349182],[0.27059805,-0.653281482,0.653281482,-0.27059805],[-1,0,-2,0],[9E+09,9E+09,9E+09,9E+09,9E+09,9E+09]];
    CONST robtarget Target_540:=[[1416.684662091,-4996.464620021,406.636213562],[0.27059805,-0.653281482,0.653281482,-0.27059805],[-1,0,-2,0],[9E+09,9E+09,9E+09,9E+09,9E+09,9E+09]];
    CONST robtarget Target_550:=[[1416.684662091,-5096.464620021,406.977213562],[0.27059805,-0.653281482,0.653281482,-0.27059805],[-1,0,-2,0],[9E+09,9E+09,9E+09,9E+09,9E+09,9E+09]];
    CONST robtarget Target_560:=[[1633.941662091,-5096.464620021,406.977213562],[0.27059805,-0.653281482,0.653281482,-0.27059805],[-1,0,-2,0],[9E+09,9E+09,9E+09,9E+09,9E+09,9E+09]];
    CONST robtarget Target_570:=[[1633.23455531,-5846.464620021,407.684320343],[0.27059805,-0.653281482,0.653281482,-0.27059805],[-1,0,-2,0],[9E+09,9E+09,9E+09,9E+09,9E+09,9E+09]];
    CONST robtarget Target_580:=[[1410.987662091,-5846.464620021,406.977213562],[0.27059805,-0.653281482,0.653281482,-0.27059805],[-1,0,-2,0],[9E+09,9E+09,9E+09,9E+09,9E+09,9E+09]];
    CONST robtarget Target_590:=[[1409.786448528,-5846.464620021,325.910427124],[0.27059805,-0.653281482,0.653281482,-0.27059805],[-1,0,-2,0],[9E+09,9E+09,9E+09,9E+09,9E+09,9E+09]];
    CONST robtarget Target_600:=[[1410.987662091,-5864.445620021,332.749213562],[0.27059805,-0.653281482,0.653281482,-0.27059805],[-1,0,-2,0],[9E+09,9E+09,9E+09,9E+09,9E+09,9E+09]];
    CONST robtarget Target_610:=[[1410.987662091,-5886.075620021,343.064213562],[0.27059805,-0.653281482,0.653281482,-0.27059805],[-1,0,-2,0],[9E+09,9E+09,9E+09,9E+09,9E+09,9E+09]];
    CONST robtarget Target_620:=[[1410.987662091,-5936.464620021,343.064213562],[0.27059805,-0.653281482,0.653281482,-0.27059805],[-1,0,-2,0],[9E+09,9E+09,9E+09,9E+09,9E+09,9E+09]];
    CONST robtarget Target_630:=[[-119.071124346,-5936.464620021,343.65],[0,-0.707106781,0.707106781,0],[-1,0,-2,0],[9E+09,9E+09,9E+09,9E+09,9E+09,9E+09]];
    CONST robtarget Target_650:=[[-117.656910783,-5846.464620021,321.414213562],[0.27059805,0.653281482,-0.653281482,-0.27059805],[-1,-1,-2,0],[9E+09,9E+09,9E+09,9E+09,9E+09,9E+09]];
    CONST robtarget Target_660:=[[-116.006910783,-5846.464620021,421.414213562],[0.27059805,0.653281482,-0.653281482,-0.27059805],[-1,-1,-2,0],[9E+09,9E+09,9E+09,9E+09,9E+09,9E+09]];
    CONST robtarget Target_670:=[[-120.833124346,-5846.464620021,430.238],[0,-0.707106781,0.707106781,0],[-1,0,-2,0],[9E+09,9E+09,9E+09,9E+09,9E+09,9E+09]];
    CONST robtarget Target_680:=[[-129.071124346,-5846.464620021,433.65],[0,-0.707106781,0.707106781,0],[-1,0,-2,0],[9E+09,9E+09,9E+09,9E+09,9E+09,9E+09]];
    CONST robtarget Target_690:=[[-619.071124346,-5846.464620021,433.65],[0,-0.707106781,0.707106781,0],[-1,0,-2,0],[9E+09,9E+09,9E+09,9E+09,9E+09,9E+09]];
    CONST robtarget Target_700:=[[-619.071124346,-4146.464620021,433.65],[0,-0.707106781,0.707106781,0],[0,0,0,0],[9E+09,9E+09,9E+09,9E+09,9E+09,9E+09]];
    CONST robtarget Target_710:=[[-129.071124346,-4146.464620021,433.65],[0,-0.707106781,0.707106781,0],[0,0,0,0],[9E+09,9E+09,9E+09,9E+09,9E+09,9E+09]];
    CONST robtarget Target_720:=[[-120.833124346,-4146.464620021,430.238],[0,-0.707106781,0.707106781,0],[0,0,0,0],[9E+09,9E+09,9E+09,9E+09,9E+09,9E+09]];
    CONST robtarget Target_730:=[[-116.006910783,-4146.464620021,421.414213562],[0.183012702,0.683012702,-0.683012702,-0.183012702],[0,0,0,0],[9E+09,9E+09,9E+09,9E+09,9E+09,9E+09]];
    CONST robtarget Target_740:=[[-117.656910783,-4146.464620021,336.414213562],[0.27059805,0.653281482,-0.653281482,-0.27059805],[0,0,0,0],[9E+09,9E+09,9E+09,9E+09,9E+09,9E+09]];
    CONST robtarget Target_750:=[[-117.656910783,-4146.464620021,321.414213562],[0.27059805,0.653281482,-0.653281482,-0.27059805],[0,0,0,0],[9E+09,9E+09,9E+09,9E+09,9E+09,9E+09]];
    CONST robtarget Target_760:=[[-117.656910783,-4127.483620021,332.749213562],[0.27059805,0.653281482,-0.653281482,-0.27059805],[0,0,0,0],[9E+09,9E+09,9E+09,9E+09,9E+09,9E+09]];
    CONST robtarget Target_770:=[[-119.071124346,-4106.853620021,343.65],[0,-0.707106781,0.707106781,0],[0,0,0,0],[9E+09,9E+09,9E+09,9E+09,9E+09,9E+09]];
    CONST robtarget Target_780:=[[-119.071124346,-4056.464620021,343.65],[0,-0.707106781,0.707106781,0],[0,0,0,0],[9E+09,9E+09,9E+09,9E+09,9E+09,9E+09]];
    CONST robtarget Target_790:=[[1410.987662091,-4056.464620021,343.064213562],[0.27059805,-0.653281482,0.653281482,-0.27059805],[0,0,0,0],[9E+09,9E+09,9E+09,9E+09,9E+09,9E+09]];
    CONST robtarget Target_800:=[[1410.987662091,-4106.853620021,343.064213562],[0.27059805,-0.653281482,0.653281482,-0.27059805],[0,0,0,0],[9E+09,9E+09,9E+09,9E+09,9E+09,9E+09]];
    CONST robtarget Target_810:=[[1411.200662091,-4146.464620021,322.496213562],[0.27059805,-0.653281482,0.653281482,-0.27059805],[0,0,0,0],[9E+09,9E+09,9E+09,9E+09,9E+09,9E+09]];
    CONST robtarget Target_820:=[[1410.987662091,-4146.464620021,406.977213562],[0.27059805,-0.653281482,0.653281482,-0.27059805],[0,0,0,0],[9E+09,9E+09,9E+09,9E+09,9E+09,9E+09]];
    CONST robtarget Target_830:=[[1633.941662091,-4146.464620021,406.977213562],[0.27059805,-0.653281482,0.653281482,-0.27059805],[0,0,0,0],[9E+09,9E+09,9E+09,9E+09,9E+09,9E+09]];
    CONST robtarget Target_850:=[[1416.684662091,-4896.464620021,406.977213562],[0.27059805,-0.653281482,0.653281482,-0.27059805],[0,0,0,0],[9E+09,9E+09,9E+09,9E+09,9E+09,9E+09]];
    CONST robtarget Target_840:=[[1633.941662091,-4896.464620021,406.977213562],[0.27059805,-0.653281482,0.653281482,-0.27059805],[0,0,0,0],[9E+09,9E+09,9E+09,9E+09,9E+09,9E+09]];
    CONST robtarget Target_640:=[[-119.071124346,-5886.075620021,343.65],[0,-0.707106781,0.707106781,0],[-1,0,-2,0],[9E+09,9E+09,9E+09,9E+09,9E+09,9E+09]];
    CONST robtarget Target_695:=[[-618.071124346,-4996.464620021,433.382050807],[0.183012702,0.683012702,-0.683012702,-0.183012702],[-1,-1,-2,0],[9E+09,9E+09,9E+09,9E+09,9E+09,9E+09]];
!***********************************************************
    !
    ! Módulo:  Module1
    !
    ! Descripción:
    !   <Introduzca la descripción aquí>
    !
    ! Autor: Alex
    !
    ! Versión: 1.0
    !
    !***********************************************************


    !***********************************************************
    !
    ! Procedimiento Main
    !
    !   Este es el punto de entrada de su programa
    !
    !***********************************************************


VAR intnum int_entradaDI; !interrupcion

    PROC main()
        Init:

CONNECT int_entradaDI WITH rutina_entrada_digital;
iSignalDI DI_interrupcion1,1,int_entradaDI;

        MoveL Target_30,v1000,z100,MyTool\WObj:=wobj0;
        SetDO FINISH,1;
        WaitDI En_Rob,1;
        WaitTime 1;
        Ajustar;
        GOTO Init;

    ENDPROC
    PROC Ajustar()
        SetDO FINISH,0;
        MoveJ Target_30,v1000,z100,MyTool\WObj:=wobj0;
        MoveJ Target_35,v400,z10,HerramientaDeCorte\WObj:=wobj0;
        MoveL Target_40,v200,z1,HerramientaDeCorte\WObj:=wobj0;
        MoveC Target_50,Target_60,v200,z1,HerramientaDeCorte\WObj:=wobj0;
        MoveC Target_70,Target_40,v200,z1,HerramientaDeCorte\WObj:=wobj0;
        MoveJ Target_75,v600,z10,HerramientaDeCorte\WObj:=wobj0;
        MoveL Target_80,v200,z1,HerramientaDeCorte\WObj:=wobj0;
        MoveC Target_90,Target_100,v200,z1,HerramientaDeCorte\WObj:=wobj0;
        MoveC Target_110,Target_80,v200,z1,HerramientaDeCorte\WObj:=wobj0;
        MoveJ Target_115,v600,z10,HerramientaDeCorte\WObj:=wobj0;
        MoveL Target_120,v200,z1,HerramientaDeCorte\WObj:=wobj0;
        MoveC Target_130,Target_140,v200,z1,HerramientaDeCorte\WObj:=wobj0;
        MoveC Target_150,Target_120,v200,z1,HerramientaDeCorte\WObj:=wobj0;
        MoveJ Target_155,v600,z10,HerramientaDeCorte\WObj:=wobj0;
        MoveL Target_160,v200,z1,HerramientaDeCorte\WObj:=wobj0;
        MoveC Target_170,Target_180,v200,z1,HerramientaDeCorte\WObj:=wobj0;
        MoveC Target_190,Target_160,v200,z1,HerramientaDeCorte\WObj:=wobj0;
        MoveJ Target_195,v600,z10,HerramientaDeCorte\WObj:=wobj0;
        MoveL Target_200,v200,z1,HerramientaDeCorte\WObj:=wobj0;
        MoveL Target_210,v200,z1,HerramientaDeCorte\WObj:=wobj0;
        MoveL Target_220,v200,z1,HerramientaDeCorte\WObj:=wobj0;
        MoveL Target_230,v200,z1,HerramientaDeCorte\WObj:=wobj0;
        MoveL Target_200,v200,z1,HerramientaDeCorte\WObj:=wobj0;
        MoveJ Target_235,v600,z10,HerramientaDeCorte\WObj:=wobj0;
        MoveL Target_240,v200,z1,HerramientaDeCorte\WObj:=wobj0;
        MoveC Target_250,Target_260,v200,z1,HerramientaDeCorte\WObj:=wobj0;
        MoveC Target_270,Target_240,v200,z1,HerramientaDeCorte\WObj:=wobj0;
        MoveJ Target_275,v600,z10,HerramientaDeCorte\WObj:=wobj0;
        MoveL Target_280,v200,z1,HerramientaDeCorte\WObj:=wobj0;
        MoveC Target_290,Target_300,v200,z1,HerramientaDeCorte\WObj:=wobj0;
        MoveC Target_310,Target_280,v200,z1,HerramientaDeCorte\WObj:=wobj0;
        MoveJ Target_325,v600,z10,HerramientaDeCorte\WObj:=wobj0;
        MoveL Target_330,v200,z1,HerramientaDeCorte\WObj:=wobj0;
        MoveC Target_340,Target_350,v200,z1,HerramientaDeCorte\WObj:=wobj0;
        MoveC Target_360,Target_330,v200,z1,HerramientaDeCorte\WObj:=wobj0;
        MoveJ Target_365,v600,z10,HerramientaDeCorte\WObj:=wobj0;
        MoveL Target_370,v200,z1,HerramientaDeCorte\WObj:=wobj0;
        MoveC Target_380,Target_390,v200,z1,HerramientaDeCorte\WObj:=wobj0;
        MoveC Target_400,Target_370,v200,z1,HerramientaDeCorte\WObj:=wobj0;
        MoveJ Target_405,v600,z10,HerramientaDeCorte\WObj:=wobj0;
        MoveL Target_410,v200,z1,HerramientaDeCorte\WObj:=wobj0;
        MoveL Target_420,v200,z1,HerramientaDeCorte\WObj:=wobj0;
        MoveL Target_430,v200,z1,HerramientaDeCorte\WObj:=wobj0;
        MoveL Target_440,v200,z1,HerramientaDeCorte\WObj:=wobj0;
        MoveL Target_410,v200,z1,HerramientaDeCorte\WObj:=wobj0;
        MoveJ Target_445,v600,z10,HerramientaDeCorte\WObj:=wobj0;
        MoveL Target_450,v200,z1,HerramientaDeCorte\WObj:=wobj0;
        MoveC Target_460,Target_470,v200,z1,HerramientaDeCorte\WObj:=wobj0;
        MoveC Target_480,Target_450,v200,z1,HerramientaDeCorte\WObj:=wobj0;
        MoveJ Target_485,v600,z10,HerramientaDeCorte\WObj:=wobj0;
        MoveL Target_490,v200,z1,HerramientaDeCorte\WObj:=wobj0;
        MoveC Target_500,Target_510,v200,z1,HerramientaDeCorte\WObj:=wobj0;
        MoveC Target_520,Target_490,v200,z1,HerramientaDeCorte\WObj:=wobj0;
        MoveJ Target_535,v600,z10,HerramientaDeCorte\WObj:=wobj0;
        MoveL Target_540,v200,z1,HerramientaDeCorte\WObj:=wobj0;
        MoveL Target_550,v200,z1,HerramientaDeCorte\WObj:=wobj0;
        MoveL Target_560,v200,z1,HerramientaDeCorte\WObj:=wobj0;
        MoveL Target_570,v200,z1,HerramientaDeCorte\WObj:=wobj0;
        MoveL Target_580,v200,z1,HerramientaDeCorte\WObj:=wobj0;
        MoveL Target_590,v200,z1,HerramientaDeCorte\WObj:=wobj0;
        MoveL Target_600,v200,z1,HerramientaDeCorte\WObj:=wobj0;
        MoveL Target_610,v200,z1,HerramientaDeCorte\WObj:=wobj0;
        MoveL Target_620,v200,z1,HerramientaDeCorte\WObj:=wobj0;
        MoveL Target_630,v200,z1,HerramientaDeCorte\WObj:=wobj0;
        MoveL Target_640,v200,z1,HerramientaDeCorte\WObj:=wobj0;
        MoveL Target_650,v200,z1,HerramientaDeCorte\WObj:=wobj0;
        MoveL Target_660,v200,z1,HerramientaDeCorte\WObj:=wobj0;
        MoveL Target_670,v200,z1,HerramientaDeCorte\WObj:=wobj0;
        MoveL Target_680,v200,z1,HerramientaDeCorte\WObj:=wobj0;
        MoveL Target_690,v200,z1,HerramientaDeCorte\WObj:=wobj0;
        MoveL Target_695,v200,z1,HerramientaDeCorte\WObj:=wobj0;
        MoveL Target_700,v200,z1,HerramientaDeCorte\WObj:=wobj0;
        MoveL Target_710,v200,z1,HerramientaDeCorte\WObj:=wobj0;
        MoveL Target_720,v200,z1,HerramientaDeCorte\WObj:=wobj0;
        MoveL Target_730,v200,z1,HerramientaDeCorte\WObj:=wobj0;
        MoveL Target_740,v200,z1,HerramientaDeCorte\WObj:=wobj0;
        MoveL Target_750,v200,z1,HerramientaDeCorte\WObj:=wobj0;
        MoveL Target_760,v200,z1,HerramientaDeCorte\WObj:=wobj0;
        MoveL Target_770,v200,z1,HerramientaDeCorte\WObj:=wobj0;
        MoveL Target_780,v200,z1,HerramientaDeCorte\WObj:=wobj0;
        MoveL Target_790,v200,z1,HerramientaDeCorte\WObj:=wobj0;
        MoveL Target_800,v200,z1,HerramientaDeCorte\WObj:=wobj0;
        MoveL Target_810,v200,z1,HerramientaDeCorte\WObj:=wobj0;
        MoveL Target_820,v200,z1,HerramientaDeCorte\WObj:=wobj0;
        MoveL Target_830,v200,z1,HerramientaDeCorte\WObj:=wobj0;
        MoveL Target_840,v200,z1,HerramientaDeCorte\WObj:=wobj0;
        MoveL Target_850,v200,z1,HerramientaDeCorte\WObj:=wobj0;
        WaitTime 1;
        SetDO FINISH,1;
        MoveL Target_30,v1000,z100,MyTool\WObj:=wobj0;
        WaitTime 5;
    ENDPROC

      TRAP rutina_entrada_digital

WHILE DI_interrupcion1=1 DO
StopMove;
ENDWHILE

StartMove;
ENDTRAP

ENDMODULE

--- Backups/Controlador_Robot2/RAPID/TASK1/PROGMOD/CalibData.mod ---
MODULE CalibData
    PERS tooldata HerramientaDeCorte:=[TRUE,[[0,0,319.427],[1,0,0,0]],[1,[0,0,1],[1,0,0,0],0,0,0]];
ENDMODULE

--- Backups/Controlador_Robot2/RAPID/TASK1/PROGMOD/Module1.mod ---
MODULE Module1
        CONST robtarget Target_5:=[[3041.012946121,-2875.846052652,447.65],[0,0.707106781,0.707106781,0],[0,0,0,0],[9E+09,9E+09,9E+09,9E+09,9E+09,9E+09]];
    CONST robtarget Target_10:=[[3041.012946121,-2875.846052652,432.65],[0,0.707106781,0.707106781,0],[0,0,-1,0],[9E+09,9E+09,9E+09,9E+09,9E+09,9E+09]];
    CONST robtarget Target_20:=[[3053.512946121,-2863.346052652,432.65],[0,0.707106781,0.707106781,0],[0,0,-1,0],[9E+09,9E+09,9E+09,9E+09,9E+09,9E+09]];
    CONST robtarget Target_30:=[[3041.012946121,-2850.846052652,432.65],[0,0.707106781,0.707106781,0],[0,0,-1,0],[9E+09,9E+09,9E+09,9E+09,9E+09,9E+09]];
    CONST robtarget Target_40:=[[3028.512946121,-2863.346052652,432.65],[0,0.707106781,0.707106781,0],[0,0,0,0],[9E+09,9E+09,9E+09,9E+09,9E+09,9E+09]];
    CONST robtarget Target_45:=[[3041.012946121,-2025.846052652,447.65],[0,0.707106781,0.707106781,0],[-1,0,-2,0],[9E+09,9E+09,9E+09,9E+09,9E+09,9E+09]];
    CONST robtarget Target_50:=[[3041.012946121,-2025.846052652,432.65],[0,0.707106781,0.707106781,0],[-1,0,-2,0],[9E+09,9E+09,9E+09,9E+09,9E+09,9E+09]];
    CONST robtarget Target_60:=[[3053.512946121,-2013.346052652,432.65],[0,0.707106781,0.707106781,0],[-1,0,-2,0],[9E+09,9E+09,9E+09,9E+09,9E+09,9E+09]];
    CONST robtarget Target_70:=[[3041.012946121,-2000.846052652,432.65],[0,0.707106781,0.707106781,0],[-1,0,-2,0],[9E+09,9E+09,9E+09,9E+09,9E+09,9E+09]];
    CONST robtarget Target_80:=[[3028.512946121,-2013.346052652,432.65],[0,0.707106781,0.707106781,0],[-1,0,-2,0],[9E+09,9E+09,9E+09,9E+09,9E+09,9E+09]];
    CONST robtarget Target_84:=[[2603.852946121,-1658.346052652,437.65],[0,0.707106781,0.707106781,0],[-1,0,-2,0],[9E+09,9E+09,9E+09,9E+09,9E+09,9E+09]];
    CONST robtarget Target_85:=[[2603.852946121,-1658.346052652,277.65],[0,0.707106781,0.707106781,0],[-1,0,-2,0],[9E+09,9E+09,9E+09,9E+09,9E+09,9E+09]];
    CONST robtarget Target_90:=[[2603.852946121,-1658.346052652,262.65],[0,0.707106781,0.707106781,0],[-1,0,-2,0],[9E+09,9E+09,9E+09,9E+09,9E+09,9E+09]];
    CONST robtarget Target_100:=[[2613.852946121,-1648.346052652,262.65],[0,0.707106781,0.707106781,0],[-1,0,-2,0],[9E+09,9E+09,9E+09,9E+09,9E+09,9E+09]];
    CONST robtarget Target_110:=[[2603.852946121,-1638.346052652,262.65],[0,0.707106781,0.707106781,0],[-1,0,-2,0],[9E+09,9E+09,9E+09,9E+09,9E+09,9E+09]];
    CONST robtarget Target_120:=[[2593.852946121,-1648.346052652,262.65],[0,0.707106781,0.707106781,0],[-1,0,-2,0],[9E+09,9E+09,9E+09,9E+09,9E+09,9E+09]];
    CONST robtarget Target_125:=[[2603.852946121,-2288.346052652,277.65],[0,0.707106781,0.707106781,0],[-1,0,-2,0],[9E+09,9E+09,9E+09,9E+09,9E+09,9E+09]];
    CONST robtarget Target_130:=[[2603.852946121,-2288.346052652,262.65],[0,0.707106781,0.707106781,0],[-1,0,-2,0],[9E+09,9E+09,9E+09,9E+09,9E+09,9E+09]];
    CONST robtarget Target_140:=[[2613.852946121,-2278.346052652,262.65],[0,0.707106781,0.707106781,0],[-1,0,-2,0],[9E+09,9E+09,9E+09,9E+09,9E+09,9E+09]];
    CONST robtarget Target_150:=[[2603.852946121,-2268.346052652,262.65],[0,0.707106781,0.707106781,0],[-1,0,-2,0],[9E+09,9E+09,9E+09,9E+09,9E+09,9E+09]];
    CONST robtarget Target_160:=[[2593.852946121,-2278.346052652,262.65],[0,0.707106781,0.707106781,0],[-1,0,-2,0],[9E+09,9E+09,9E+09,9E+09,9E+09,9E+09]];
    CONST robtarget Target_164:=[[2603.852946121,-2288.346052652,347.65],[0,0.707106781,0.707106781,0],[-1,0,-2,0],[9E+09,9E+09,9E+09,9E+09,9E+09,9E+09]];
    CONST robtarget Target_165:=[[2592.880946121,-2374.172052652,347.65],[0,0.707106781,0.707106781,0],[-1,0,-2,0],[9E+09,9E+09,9E+09,9E+09,9E+09,9E+09]];
    CONST robtarget Target_170:=[[2592.880946121,-2374.172052652,332.65],[0,0.707106781,0.707106781,0],[-1,0,-2,0],[9E+09,9E+09,9E+09,9E+09,9E+09,9E+09]];
    CONST robtarget Target_180:=[[2191.191946121,-2374.172052652,332.65],[0,0.707106781,0.707106781,0],[-1,0,-2,0],[9E+09,9E+09,9E+09,9E+09,9E+09,9E+09]];
    CONST robtarget Target_190:=[[2191.191946121,-2502.520052652,332.65],[0,0.707106781,0.707106781,0],[0,0,0,0],[9E+09,9E+09,9E+09,9E+09,9E+09,9E+09]];
    CONST robtarget Target_200:=[[2592.880946121,-2502.520052652,332.65],[0,0.707106781,0.707106781,0],[0,0,0,0],[9E+09,9E+09,9E+09,9E+09,9E+09,9E+09]];
    CONST robtarget Target_204:=[[2603.852946121,-2608.346052652,347.65],[0,0.707106781,0.707106781,0],[0,0,0,0],[9E+09,9E+09,9E+09,9E+09,9E+09,9E+09]];
    CONST robtarget Target_205:=[[2603.852946121,-2608.346052652,277.65],[0,0.707106781,0.707106781,0],[0,0,0,0],[9E+09,9E+09,9E+09,9E+09,9E+09,9E+09]];
    CONST robtarget Target_210:=[[2603.852946121,-2608.346052652,262.65],[0,0.707106781,0.707106781,0],[0,0,0,0],[9E+09,9E+09,9E+09,9E+09,9E+09,9E+09]];
    CONST robtarget Target_220:=[[2613.852946121,-2598.346052652,262.65],[0,0.707106781,0.707106781,0],[0,0,0,0],[9E+09,9E+09,9E+09,9E+09,9E+09,9E+09]];
    CONST robtarget Target_230:=[[2603.852946121,-2588.346052652,262.65],[0,0.707106781,0.707106781,0],[0,0,0,0],[9E+09,9E+09,9E+09,9E+09,9E+09,9E+09]];
    CONST robtarget Target_240:=[[2593.852946121,-2598.346052652,262.65],[0,0.707106781,0.707106781,0],[0,0,0,0],[9E+09,9E+09,9E+09,9E+09,9E+09,9E+09]];
    CONST robtarget Target_245:=[[2603.852946121,-3238.346052652,277.65],[0,0.707106781,0.707106781,0],[0,0,0,0],[9E+09,9E+09,9E+09,9E+09,9E+09,9E+09]];
    CONST robtarget Target_250:=[[2603.852946121,-3238.346052652,262.65],[0,0.707106781,0.707106781,0],[0,0,0,0],[9E+09,9E+09,9E+09,9E+09,9E+09,9E+09]];
    CONST robtarget Target_260:=[[2613.852946121,-3228.346052652,262.65],[0,0.707106781,0.707106781,0],[0,0,0,0],[9E+09,9E+09,9E+09,9E+09,9E+09,9E+09]];
    CONST robtarget Target_270:=[[2603.852946121,-3218.346052652,262.65],[0,0.707106781,0.707106781,0],[0,0,0,0],[9E+09,9E+09,9E+09,9E+09,9E+09,9E+09]];
    CONST robtarget Target_280:=[[2593.852946121,-3228.346052652,262.65],[0,0.707106781,0.707106781,0],[0,0,0,0],[9E+09,9E+09,9E+09,9E+09,9E+09,9E+09]];
    CONST robtarget Target_284:=[[2603.852946121,-3238.346052652,317.65],[0,0.707106781,0.707106781,0],[0,0,0,0],[9E+09,9E+09,9E+09,9E+09,9E+09,9E+09]];
    CONST robtarget Target_285:=[[2153.852946121,-3238.346052652,327.65],[0,0.707106781,0.707106781,0],[0,0,0,0],[9E+09,9E+09,9E+09,9E+09,9E+09,9E+09]];
    CONST robtarget Target_290:=[[2153.852946121,-3238.346052652,312.65],[0,0.707106781,0.707106781,0],[0,0,0,0],[9E+09,9E+09,9E+09,9E+09,9E+09,9E+09]];
    CONST robtarget Target_300:=[[2163.852946121,-3228.346052652,312.65],[0,0.707106781,0.707106781,0],[0,0,0,0],[9E+09,9E+09,9E+09,9E+09,9E+09,9E+09]];
    CONST robtarget Target_310:=[[2153.852946121,-3218.346052652,312.65],[0,0.707106781,0.707106781,0],[0,0,0,0],[9E+09,9E+09,9E+09,9E+09,9E+09,9E+09]];
    CONST robtarget Target_320:=[[2143.852946121,-3228.346052652,312.65],[0,0.707106781,0.707106781,0],[0,0,0,0],[9E+09,9E+09,9E+09,9E+09,9E+09,9E+09]];
    CONST robtarget Target_325:=[[2153.852946121,-2608.346052652,327.65],[0,0.707106781,0.707106781,0],[0,0,0,0],[9E+09,9E+09,9E+09,9E+09,9E+09,9E+09]];
    CONST robtarget Target_330:=[[2153.852946121,-2608.346052652,312.65],[0,0.707106781,0.707106781,0],[0,0,0,0],[9E+09,9E+09,9E+09,9E+09,9E+09,9E+09]];
    CONST robtarget Target_340:=[[2163.852946121,-2598.346052652,312.65],[0,0.707106781,0.707106781,0],[0,0,0,0],[9E+09,9E+09,9E+09,9E+09,9E+09,9E+09]];
    CONST robtarget Target_350:=[[2153.852946121,-2588.346052652,312.65],[0,0.707106781,0.707106781,0],[0,0,0,0],[9E+09,9E+09,9E+09,9E+09,9E+09,9E+09]];
    CONST robtarget Target_360:=[[2143.852946121,-2598.346052652,312.65],[0,0.707106781,0.707106781,0],[0,0,0,0],[9E+09,9E+09,9E+09,9E+09,9E+09,9E+09]];
    CONST robtarget Target_364:=[[2153.852946121,-2608.346052652,357.65],[0,0.707106781,0.707106781,0],[0,0,0,0],[9E+09,9E+09,9E+09,9E+09,9E+09,9E+09]];
    CONST robtarget Target_365:=[[2071.138946121,-2483.346052652,349.903],[0,0.707106781,0.707106781,0],[0,0,0,0],[9E+09,9E+09,9E+09,9E+09,9E+09,9E+09]];
    CONST robtarget Target_370:=[[2071.138946121,-2483.346052652,334.903],[0,0.707106781,0.707106781,0],[0,0,0,0],[9E+09,9E+09,9E+09,9E+09,9E+09,9E+09]];
    CONST robtarget Target_380:=[[2071.138946121,-2393.346052652,334.903],[0,0.707106781,0.707106781,0],[0,0,0,0],[9E+09,9E+09,9E+09,9E+09,9E+09,9E+09]];
    CONST robtarget Target_390:=[[1871.138946121,-2393.346052652,345.449],[0,0.707106781,0.707106781,0],[0,0,0,0],[9E+09,9E+09,9E+09,9E+09,9E+09,9E+09]];
    CONST robtarget Target_400:=[[1871.138946121,-2483.346052652,345.449],[0,0.707106781,0.707106781,0],[0,0,0,0],[9E+09,9E+09,9E+09,9E+09,9E+09,9E+09]];
    CONST robtarget Target_414:=[[2153.852946121,-2288.346052652,357.65],[0,0.707106781,0.707106781,0],[-1,0,-2,0],[9E+09,9E+09,9E+09,9E+09,9E+09,9E+09]];
    CONST robtarget Target_415:=[[2153.852946121,-2288.346052652,327.65],[0,0.707106781,0.707106781,0],[-1,0,-2,0],[9E+09,9E+09,9E+09,9E+09,9E+09,9E+09]];
    CONST robtarget Target_430:=[[2153.852946121,-2288.346052652,312.65],[0,0.707106781,0.707106781,0],[-1,0,-2,0],[9E+09,9E+09,9E+09,9E+09,9E+09,9E+09]];
    CONST robtarget Target_440:=[[2163.852946121,-2278.346052652,312.65],[0,0.707106781,0.707106781,0],[-1,0,-2,0],[9E+09,9E+09,9E+09,9E+09,9E+09,9E+09]];
    CONST robtarget Target_450:=[[2153.852946121,-2268.346052652,312.65],[0,0.707106781,0.707106781,0],[-1,0,-2,0],[9E+09,9E+09,9E+09,9E+09,9E+09,9E+09]];
    CONST robtarget Target_460:=[[2143.852946121,-2278.346052652,312.65],[0,0.707106781,0.707106781,0],[-1,0,-2,0],[9E+09,9E+09,9E+09,9E+09,9E+09,9E+09]];
    CONST robtarget Target_465:=[[2153.852946121,-1658.346052652,327.65],[0,0.707106781,0.707106781,0],[-1,0,-2,0],[9E+09,9E+09,9E+09,9E+09,9E+09,9E+09]];
    CONST robtarget Target_470:=[[2153.852946121,-1658.346052652,312.65],[0,0.707106781,0.707106781,0],[-1,0,-2,0],[9E+09,9E+09,9E+09,9E+09,9E+09,9E+09]];
    CONST robtarget Target_480:=[[2163.852946121,-1648.346052652,312.65],[0,0.707106781,0.707106781,0],[-1,0,-2,0],[9E+09,9E+09,9E+09,9E+09,9E+09,9E+09]];
    CONST robtarget Target_490:=[[2153.852946121,-1638.346052652,312.65],[0,0.707106781,0.707106781,0],[-1,0,-2,0],[9E+09,9E+09,9E+09,9E+09,9E+09,9E+09]];
    CONST robtarget Target_500:=[[2143.852946121,-1648.346052652,311.65],[0,0.707106781,0.707106781,0],[-1,0,-2,0],[9E+09,9E+09,9E+09,9E+09,9E+09,9E+09]];
    CONST robtarget Target_515:=[[1450.826081749,-2438.346052652,419.36513562],[0.27059805,-0.653281482,-0.653281482,0.27059805],[0,0,0,0],[9E+09,9E+09,9E+09,9E+09,9E+09,9E+09]];
    CONST robtarget Target_520:=[[1438.098159684,-2438.346052652,406.637213562],[0.27059805,-0.653281482,-0.653281482,0.27059805],[0,0,0,0],[9E+09,9E+09,9E+09,9E+09,9E+09,9E+09]];
    CONST robtarget Target_530:=[[1438.098159684,-2338.346052652,406.977213562],[0.27059805,-0.653281482,-0.653281482,0.27059805],[-1,0,-2,0],[9E+09,9E+09,9E+09,9E+09,9E+09,9E+09]];
    CONST robtarget Target_540:=[[1220.840159684,-2338.346052652,406.977213562],[0.27059805,-0.653281482,-0.653281482,0.27059805],[-1,0,-2,0],[9E+09,9E+09,9E+09,9E+09,9E+09,9E+09]];
    CONST robtarget Target_550:=[[1220.840159684,-1588.346052652,406.977213562],[0.27059805,-0.653281482,-0.653281482,0.27059805],[-1,0,-2,0],[9E+09,9E+09,9E+09,9E+09,9E+09,9E+09]];
    CONST robtarget Target_560:=[[1443.794159684,-1588.346052652,406.977213562],[0.27059805,-0.653281482,-0.653281482,0.27059805],[-1,0,-2,0],[9E+09,9E+09,9E+09,9E+09,9E+09,9E+09]];
    CONST robtarget Target_570:=[[1444.288266465,-1588.346052652,323.203320343],[0.27059805,-0.653281482,-0.653281482,0.27059805],[-1,0,-2,0],[9E+09,9E+09,9E+09,9E+09,9E+09,9E+09]];
    CONST robtarget Target_580:=[[1443.794159684,-1569.365052652,332.749213562],[0.27059805,-0.653281482,-0.653281482,0.27059805],[-1,0,-2,0],[9E+09,9E+09,9E+09,9E+09,9E+09,9E+09]];
    CONST robtarget Target_590:=[[1443.794159684,-1548.735052652,343.064213562],[0.27059805,-0.653281482,-0.653281482,0.27059805],[-1,0,-2,0],[9E+09,9E+09,9E+09,9E+09,9E+09,9E+09]];
    CONST robtarget Target_600:=[[1443.794159684,-1523.541052652,343.064213562],[0.27059805,-0.653281482,-0.653281482,0.27059805],[-1,0,-2,0],[9E+09,9E+09,9E+09,9E+09,9E+09,9E+09]];
    CONST robtarget Target_610:=[[1443.794159684,-1498.346052652,343.064213562],[0.27059805,-0.653281482,-0.653281482,0.27059805],[-1,0,-2,0],[9E+09,9E+09,9E+09,9E+09,9E+09,9E+09]];
    CONST robtarget Target_620:=[[2973.852946121,-1498.346052652,343.65],[0,0.707106781,0.707106781,0],[-1,0,-2,0],[9E+09,9E+09,9E+09,9E+09,9E+09,9E+09]];
    CONST robtarget Target_630:=[[2973.852946121,-1548.735052652,343.65],[0,0.707106781,0.707106781,0],[-1,0,-2,0],[9E+09,9E+09,9E+09,9E+09,9E+09,9E+09]];
    CONST robtarget Target_640:=[[2972.438732558,-1569.365052652,332.749213562],[0.27059805,0.653281482,0.653281482,0.27059805],[-1,-1,-2,0],[9E+09,9E+09,9E+09,9E+09,9E+09,9E+09]];
    CONST robtarget Target_650:=[[2971.024518995,-1588.346052652,322.828427124],[0.27059805,0.653281482,0.653281482,0.27059805],[-1,-1,-2,0],[9E+09,9E+09,9E+09,9E+09,9E+09,9E+09]];
    CONST robtarget Target_660:=[[2971.202946121,-1588.346052652,421.732050807],[0.183012702,0.683012702,0.683012702,0.183012702],[-1,-1,-2,0],[9E+09,9E+09,9E+09,9E+09,9E+09,9E+09]];
    CONST robtarget Target_670:=[[2974.614946121,-1588.346052652,429.970050807],[0.183012702,0.683012702,0.683012702,0.183012702],[-1,-1,-2,0],[9E+09,9E+09,9E+09,9E+09,9E+09,9E+09]];
    CONST robtarget Target_680:=[[2983.852946121,-1588.346052652,433.65],[0,0.707106781,0.707106781,0],[-1,0,-2,0],[9E+09,9E+09,9E+09,9E+09,9E+09,9E+09]];
    CONST robtarget Target_700:=[[3473.852946121,-1588.346052652,433.65],[0,0.707106781,0.707106781,0],[-1,0,-2,0],[9E+09,9E+09,9E+09,9E+09,9E+09,9E+09]];
    CONST robtarget Target_710:=[[3472.852946116,-2438.346052652,433.382050805],[0.183012703,0.683012702,0.683012702,0.183012703],[0,0,0,0],[9E+09,9E+09,9E+09,9E+09,9E+09,9E+09]];
    CONST robtarget Target_720:=[[3473.852946121,-3288.346052652,433.65],[0,0.707106781,0.707106781,0],[0,0,0,0],[9E+09,9E+09,9E+09,9E+09,9E+09,9E+09]];
    CONST robtarget Target_730:=[[2983.852946121,-3288.346052652,433.65],[0,0.707106781,0.707106781,0],[0,0,0,0],[9E+09,9E+09,9E+09,9E+09,9E+09,9E+09]];
    CONST robtarget Target_740:=[[2974.614946121,-3288.346052652,429.970050807],[0.183012702,0.683012702,0.683012702,0.183012702],[0,0,0,0],[9E+09,9E+09,9E+09,9E+09,9E+09,9E+09]];
    CONST robtarget Target_750:=[[2970.788732558,-3288.346052652,421.414213562],[0.183012702,0.683012702,0.683012702,0.183012702],[0,0,0,0],[9E+09,9E+09,9E+09,9E+09,9E+09,9E+09]];
    CONST robtarget Target_760:=[[2971.024518995,-3288.346052652,322.828427124],[0.27059805,0.653281482,0.653281482,0.27059805],[0,0,0,0],[9E+09,9E+09,9E+09,9E+09,9E+09,9E+09]];
    CONST robtarget Target_770:=[[2972.438732558,-3307.327052652,332.749213562],[0.27059805,0.653281482,0.653281482,0.27059805],[0,0,0,0],[9E+09,9E+09,9E+09,9E+09,9E+09,9E+09]];
    CONST robtarget Target_780:=[[2973.852946121,-3327.957052652,343.65],[0,0.707106781,0.707106781,0],[0,0,0,0],[9E+09,9E+09,9E+09,9E+09,9E+09,9E+09]];
    CONST robtarget Target_790:=[[2973.852946121,-3378.346052652,343.65],[0,0.707106781,0.707106781,0],[0,0,0,0],[9E+09,9E+09,9E+09,9E+09,9E+09,9E+09]];
    CONST robtarget Target_800:=[[1443.794159684,-3378.346052652,343.064213562],[0.27059805,-0.653281482,-0.653281482,0.27059805],[0,0,0,0],[9E+09,9E+09,9E+09,9E+09,9E+09,9E+09]];
    CONST robtarget Target_810:=[[1443.794159684,-3327.957052652,343.064213562],[0.27059805,-0.653281482,-0.653281482,0.27059805],[0,0,0,0],[9E+09,9E+09,9E+09,9E+09,9E+09,9E+09]];
    CONST robtarget Target_820:=[[1444.288266465,-3288.346052652,323.203320343],[0.27059805,-0.653281482,-0.653281482,0.27059805],[0,0,0,0],[9E+09,9E+09,9E+09,9E+09,9E+09,9E+09]];
    CONST robtarget Target_830:=[[1443.581159684,-3288.346052652,406.977213562],[0.27059805,-0.653281482,-0.653281482,0.27059805],[0,0,0,0],[9E+09,9E+09,9E+09,9E+09,9E+09,9E+09]];
    CONST robtarget Target_840:=[[1221.157996929,-3288.346052652,406.562999999],[0.353553391,-0.612372436,-0.612372436,0.353553391],[0,0,0,0],[9E+09,9E+09,9E+09,9E+09,9E+09,9E+09]];
    CONST robtarget Target_850:=[[1220.840159684,-2538.346052652,406.977213562],[0.27059805,-0.653281482,-0.653281482,0.27059805],[0,0,0,0],[9E+09,9E+09,9E+09,9E+09,9E+09,9E+09]];
    CONST robtarget Target_860:=[[1438.098159684,-2538.346052652,406.977213562],[0.27059805,-0.653281482,-0.653281482,0.27059805],[0,0,0,0],[9E+09,9E+09,9E+09,9E+09,9E+09,9E+09]];
    CONST robtarget Home:=[[2523.400603118,-2378.132052652,3271.543828966],[0,-0.661802163,0,0.749678529],[0,0,0,0],[9E+09,9E+09,9E+09,9E+09,9E+09,9E+09]];
!***********************************************************
    !
    ! Módulo:  Module1
    !
    ! Descripción:
    !   <Introduzca la descripción aquí>
    !
    ! Autor: Alex
    !
    ! Versión: 1.0
    !
    !***********************************************************


    !***********************************************************
    !
    ! Procedimiento Main
    !
    !   Este es el punto de entrada de su programa
    !
    !***********************************************************


VAR intnum int_entradaDI; !interrupcion

    PROC main()
        Init:

CONNECT int_entradaDI WITH rutina_entrada_digital;
iSignalDI DI_interrupcion2,1,int_entradaDI;

        MoveJ Home,v1000,z100,HerramientaDeCorte\WObj:=wobj0;
        SetDO FINISH,1;
        WaitDI En_Rob,1;
        WaitTime 1;
        Path_10;
        GOTO Init;
    ENDPROC
    PROC Path_10()
        SetDO FINISH,0;
        MoveJ Target_5,v600,z10,HerramientaDeCorte\WObj:=wobj0;
        MoveL Target_10,v1000,z100,HerramientaDeCorte\WObj:=wobj0;
        MoveC Target_20,Target_30,v1000,z100,HerramientaDeCorte\WObj:=wobj0;
        MoveC Target_40,Target_10,v1000,z100,HerramientaDeCorte\WObj:=wobj0;
        MoveJ Target_5,v600,z10,HerramientaDeCorte\WObj:=wobj0;
        MoveJ Target_45,v600,z10,HerramientaDeCorte\WObj:=wobj0;
        MoveL Target_50,v1000,z100,HerramientaDeCorte\WObj:=wobj0;
        MoveC Target_60,Target_70,v1000,z100,HerramientaDeCorte\WObj:=wobj0;
        MoveC Target_80,Target_50,v1000,z100,HerramientaDeCorte\WObj:=wobj0;
        MoveJ Target_45,v600,z10,HerramientaDeCorte\WObj:=wobj0;
        MoveJ Target_84,v600,z10,HerramientaDeCorte\WObj:=wobj0;
        MoveJ Target_85,v600,z10,HerramientaDeCorte\WObj:=wobj0;
        MoveL Target_90,v1000,z100,HerramientaDeCorte\WObj:=wobj0;
        MoveC Target_100,Target_110,v1000,z100,HerramientaDeCorte\WObj:=wobj0;
        MoveC Target_120,Target_90,v1000,z100,HerramientaDeCorte\WObj:=wobj0;
        MoveJ Target_85,v600,z10,HerramientaDeCorte\WObj:=wobj0;
        MoveJ Target_125,v600,z10,HerramientaDeCorte\WObj:=wobj0;
        MoveL Target_130,v1000,z100,HerramientaDeCorte\WObj:=wobj0;
        MoveC Target_140,Target_150,v1000,z100,HerramientaDeCorte\WObj:=wobj0;
        MoveC Target_160,Target_130,v1000,z100,HerramientaDeCorte\WObj:=wobj0;
        MoveJ Target_125,v600,z10,HerramientaDeCorte\WObj:=wobj0;
        MoveJ Target_164,v600,z10,HerramientaDeCorte\WObj:=wobj0;
        MoveJ Target_165,v600,z10,HerramientaDeCorte\WObj:=wobj0;
        MoveL Target_170,v1000,z100,HerramientaDeCorte\WObj:=wobj0;
        MoveL Target_180,v200,z1,HerramientaDeCorte\WObj:=wobj0;
        MoveL Target_190,v200,z1,HerramientaDeCorte\WObj:=wobj0;
        MoveL Target_200,v200,z1,HerramientaDeCorte\WObj:=wobj0;
        MoveL Target_170,v200,z1,HerramientaDeCorte\WObj:=wobj0;
        MoveJ Target_165,v600,z10,HerramientaDeCorte\WObj:=wobj0;
        MoveJ Target_204,v600,z10,HerramientaDeCorte\WObj:=wobj0;
        MoveJ Target_205,v600,z10,HerramientaDeCorte\WObj:=wobj0;
        MoveL Target_210,v1000,z100,HerramientaDeCorte\WObj:=wobj0;
        MoveC Target_220,Target_230,v1000,z100,HerramientaDeCorte\WObj:=wobj0;
        MoveC Target_240,Target_210,v1000,z100,HerramientaDeCorte\WObj:=wobj0;
        MoveJ Target_205,v600,z10,HerramientaDeCorte\WObj:=wobj0;
        MoveJ Target_245,v600,z10,HerramientaDeCorte\WObj:=wobj0;
        MoveL Target_250,v1000,z100,HerramientaDeCorte\WObj:=wobj0;
        MoveC Target_260,Target_270,v1000,z100,HerramientaDeCorte\WObj:=wobj0;
        MoveC Target_280,Target_250,v1000,z100,HerramientaDeCorte\WObj:=wobj0;
        MoveJ Target_245,v600,z10,HerramientaDeCorte\WObj:=wobj0;
        MoveJ Target_284,v600,z10,HerramientaDeCorte\WObj:=wobj0;
        MoveJ Target_285,v600,z10,HerramientaDeCorte\WObj:=wobj0;
        MoveL Target_290,v1000,z100,HerramientaDeCorte\WObj:=wobj0;
        MoveC Target_300,Target_310,v1000,z100,HerramientaDeCorte\WObj:=wobj0;
        MoveC Target_320,Target_290,v1000,z100,HerramientaDeCorte\WObj:=wobj0;
        MoveJ Target_285,v600,z10,HerramientaDeCorte\WObj:=wobj0;
        MoveJ Target_325,v600,z10,HerramientaDeCorte\WObj:=wobj0;
        MoveL Target_330,v1000,z100,HerramientaDeCorte\WObj:=wobj0;
        MoveC Target_340,Target_350,v1000,z100,HerramientaDeCorte\WObj:=wobj0;
        MoveC Target_360,Target_330,v1000,z100,HerramientaDeCorte\WObj:=wobj0;
        MoveJ Target_364,v600,z10,HerramientaDeCorte\WObj:=wobj0;
        MoveJ Target_365,v600,z10,HerramientaDeCorte\WObj:=wobj0;
        MoveL Target_370,v400,z1,HerramientaDeCorte\WObj:=wobj0;
        MoveL Target_380,v400,z1,HerramientaDeCorte\WObj:=wobj0;
        MoveL Target_390,v400,z1,HerramientaDeCorte\WObj:=wobj0;
        MoveL Target_400,v400,z1,HerramientaDeCorte\WObj:=wobj0;
        MoveL Target_370,v400,z1,HerramientaDeCorte\WObj:=wobj0;
        MoveJ Target_365,v600,z10,HerramientaDeCorte\WObj:=wobj0;
        MoveJ Target_414,v600,z10,HerramientaDeCorte\WObj:=wobj0;
        MoveJ Target_415,v600,z10,HerramientaDeCorte\WObj:=wobj0;
        MoveL Target_430,v1000,z100,HerramientaDeCorte\WObj:=wobj0;
        MoveC Target_440,Target_450,v1000,z100,HerramientaDeCorte\WObj:=wobj0;
        MoveC Target_460,Target_430,v1000,z100,HerramientaDeCorte\WObj:=wobj0;
        MoveJ Target_415,v600,z10,HerramientaDeCorte\WObj:=wobj0;
        MoveJ Target_465,v600,z10,HerramientaDeCorte\WObj:=wobj0;
        MoveL Target_470,v1000,z100,HerramientaDeCorte\WObj:=wobj0;
        MoveC Target_480,Target_490,v1000,z100,HerramientaDeCorte\WObj:=wobj0;
        MoveC Target_500,Target_470,v1000,z100,HerramientaDeCorte\WObj:=wobj0;
        MoveJ Target_465,v600,z10,HerramientaDeCorte\WObj:=wobj0;
        MoveJ Target_515,v600,z10,HerramientaDeCorte\WObj:=wobj0;
        MoveL Target_520,v200,z1,HerramientaDeCorte\WObj:=wobj0;
        MoveL Target_530,v200,z1,HerramientaDeCorte\WObj:=wobj0;
        MoveL Target_540,v200,z1,HerramientaDeCorte\WObj:=wobj0;
        MoveL Target_550,v200,z1,HerramientaDeCorte\WObj:=wobj0;
        MoveL Target_560,v200,z1,HerramientaDeCorte\WObj:=wobj0;
        MoveL Target_570,v200,z1,HerramientaDeCorte\WObj:=wobj0;
        MoveL Target_580,v200,z1,HerramientaDeCorte\WObj:=wobj0;
        MoveL Target_590,v200,z1,HerramientaDeCorte\WObj:=wobj0;
        MoveL Target_600,v200,z1,HerramientaDeCorte\WObj:=wobj0;
        MoveL Target_610,v200,z1,HerramientaDeCorte\WObj:=wobj0;
        MoveL Target_620,v200,z1,HerramientaDeCorte\WObj:=wobj0;
        MoveL Target_630,v200,z1,HerramientaDeCorte\WObj:=wobj0;
        MoveL Target_640,v200,z1,HerramientaDeCorte\WObj:=wobj0;
        MoveL Target_650,v200,z1,HerramientaDeCorte\WObj:=wobj0;
        MoveL Target_660,v200,z1,HerramientaDeCorte\WObj:=wobj0;
        MoveL Target_670,v200,z1,HerramientaDeCorte\WObj:=wobj0;
        MoveL Target_680,v200,z1,HerramientaDeCorte\WObj:=wobj0;
        MoveL Target_700,v200,z1,HerramientaDeCorte\WObj:=wobj0;
        MoveL Target_710,v200,z1,HerramientaDeCorte\WObj:=wobj0;
        MoveL Target_720,v200,z1,HerramientaDeCorte\WObj:=wobj0;
        MoveL Target_730,v200,z1,HerramientaDeCorte\WObj:=wobj0;
        MoveL Target_740,v200,z1,HerramientaDeCorte\WObj:=wobj0;
        MoveL Target_750,v200,z1,HerramientaDeCorte\WObj:=wobj0;
        MoveL Target_760,v200,z1,HerramientaDeCorte\WObj:=wobj0;
        MoveL Target_770,v200,z1,HerramientaDeCorte\WObj:=wobj0;
        MoveL Target_780,v200,z1,HerramientaDeCorte\WObj:=wobj0;
        MoveL Target_790,v200,z1,HerramientaDeCorte\WObj:=wobj0;
        MoveL Target_800,v200,z1,HerramientaDeCorte\WObj:=wobj0;
        MoveL Target_810,v200,z1,HerramientaDeCorte\WObj:=wobj0;
        MoveL Target_820,v200,z1,HerramientaDeCorte\WObj:=wobj0;
        MoveL Target_830,v200,z1,HerramientaDeCorte\WObj:=wobj0;
        MoveL Target_840,v200,z1,HerramientaDeCorte\WObj:=wobj0;
        MoveL Target_850,v200,z1,HerramientaDeCorte\WObj:=wobj0;
        MoveL Target_860,v200,z1,HerramientaDeCorte\WObj:=wobj0;
        WaitTime 1;
        SetDO FINISH,1;
        MoveJ Home,v1000,z100,HerramientaDeCorte\WObj:=wobj0;
        WaitTime 5;
    ENDPROC
          TRAP rutina_entrada_digital

WHILE DI_interrupcion2=1 DO
StopMove;
ENDWHILE

StartMove;
ENDTRAP

ENDMODULE

--- Backups/Controlador_PickPlace/SYSPAR/EIO.cfg ---
EIO:CFG_1.0:6:1::
#
EIO_SIGNAL:

      -Name "V_ON" -SignalType "DO"\
      -Label "Enables the attach action from band1 to robots"

      -Name "V_Out1" -SignalType "DO"\
      -Label "Enables the deattach action for stage 1"

      -Name "Rob_ON" -SignalType "DI" -Label "Reads the signal of sensor 1"

      -Name "Rob_ON1" -SignalType "DI"\
      -Label "Enables pick and place from band to stage 1"

      -Name "Rob_ON2" -SignalType "DI"\
      -Label "Enables pick and place from band to stage 2"

      -Name "V_ON1" -SignalType "DO"\
      -Label "Enables the attach from robot 1 to band 2"

      -Name "V_ON2" -SignalType "DO"\
      -Label "Enables the attach from robot 2 to band 2"

      -Name "V_Out2" -SignalType "DO"\
      -Label "Enables the deattach action for stage 2"

      -Name "V_Out" -SignalType "DO"\
      -Label "Enables the deattach action for stages"

      -Name "Pick_1" -SignalType "DI"\
      -Label "Enables pick and place from stage 1 to table"

      -Name "Pick_2" -SignalType "DI"\
      -Label "Enables pick and place from stage 2 to table"

      -Name "U_Rob1" -SignalType "DO"\
      -Label "Unables the robot 1 after picking the piece of the stage"

      -Name "U_Rob2" -SignalType "DO"\
      -Label "Unables the robot 2 after picking the piece of the stage"

--- Backups/Controlador_Robot1/SYSPAR/EIO.cfg ---
EIO:CFG_1.0:6:1::
#
EIO_SIGNAL:

      -Name "En_Rob" -SignalType "DI"\
      -Label "Robots starts to work when carpet is set"

      -Name "FINISH" -SignalType "DO" -Label "Is on when Robot finish cutting"

      -Name "U_Rob" -SignalType "DI"\
      -Label "Unables the robot while package is taken"

      -Name "Unable" -SignalType "DO"\
      -Label "Stops the robot once finishes cutting"

      -Name "DI_interrupcion1" -SignalType "DI"\
      -Label "Habilita la interrupción del robot 1"

      -Name "DI_interrupcion2" -SignalType "DI"\
      -Label "Interrupción del robot 2"

--- Backups/Controlador_Robot2/SYSPAR/EIO.cfg ---
EIO:CFG_1.0:6:1::
#
EIO_SIGNAL:

      -Name "FINISH" -SignalType "DO" -Label "On when robot is not cutting"

      -Name "En_Rob" -SignalType "DI"\
      -Label "Enables the robot and start trajectory"

      -Name "U_Rob" -SignalType "DI"\
      -Label "Unables the robot while package is taken"

      -Name "Unable" -SignalType "DO"\
      -Label "Stops the robot once finishes cutting"

      -Name "DI_interrupcion2" -SignalType "DI"\
      -Label "Habilita la interrupcion del motor 2"
